LIN {X 0,Y 434.581,Z 927.636,A -85,B 0,C 180,E1 8882.861,E2 8882.861} C_VEL
LIN {X 0,Y 430.893,Z 955.392,A -85,B 0,C 180,E1 8887.344,E2 8887.344} C_VEL
LIN {X 0,Y 428.364,Z 976.944,A -85,B 0,C 180,E1 8892.013,E2 8892.013} C_VEL
LIN {X 0,Y 426.942,Z 993.408,A -85,B 0,C 180,E1 8896.966,E2 8896.966} C_VEL
LIN {X 0,Y 426.344,Z 1004.121,A -85,B 0,C 180,E1 8901.864,E2 8901.864} C_VEL
LIN {X 0,Y 426.1,Z 1008.94,A -85,B 0,C 180,E1 8905.941,E2 8905.941} C_VEL
LIN {X 0,Y 426.135,Z 1010.5,A -85,B 0,C 180,E1 8910.003,E2 8910.003} C_VEL
LIN {X 0,Y 426.114,Z 1008.916,A -85,B 0,C 180,E1 8914.065,E2 8914.065} C_VEL
LIN {X 0,Y 426.347,Z 1004.111,A -85,B 0,C 180,E1 8918.143,E2 8918.143} C_VEL
LIN {X 0,Y 427.008,Z 993.215,A -85,B 0,C 180,E1 8923.05,E2 8923.05} C_VEL
LIN {X 0,Y 428.484,Z 976.134,A -85,B 0,C 180,E1 8928.036,E2 8928.036} C_VEL
LIN {X 0,Y 430.871,Z 953.792,A -85,B 0,C 180,E1 8932.663,E2 8932.663} C_VEL
LIN {X 0,Y 434.231,Z 925.274,A -85,B 0,C 180,E1 8937.015,E2 8937.015} C_VEL
LIN {X 0,Y 438.15,Z 892.411,A -85,B 0,C 180,E1 8940.744,E2 8940.744} C_VEL
LIN {X 0,Y 442.235,Z 855.915,A -85,B 0,C 180,E1 8943.828,E2 8943.828} C_VEL
LIN {X 0,Y 446.217,Z 814.757,A -85,B 0,C 180,E1 8946.335,E2 8946.335} C_VEL
LIN {X 0,Y 449.648,Z 772.764,A -85,B 0,C 180,E1 8948.036,E2 8948.036} C_VEL
LIN {X 0,Y 450.402,Z 750.353,A -85,B 0,C 180,E1 8948.691,E2 8948.691} C_VEL
LIN {X 0,Y 439.584,Z 726.546,A -85,B 0,C 180,E1 8950.23,E2 8950.23} C_VEL
LIN {X 0,Y 430.713,Z 701.682,A -85,B 0,C 180,E1 8951.883,E2 8951.883} C_VEL
LIN {X 0,Y 424.876,Z 685.03,A -85,B 0,C 180,E1 8954.111,E2 8954.111} C_VEL
LIN {X 0,Y 424.882,Z 685.03,A -85,B 0,C 180,E1 8960.26,E2 8960.26} C_VEL
LIN {X 0,Y 424.85,Z 685.03,A -85,B 0,C 180,E1 8965.366,E2 8965.366} C_VEL
LIN {X 0,Y 424.908,Z 685.03,A -85,B 0,C 180,E1 8970.183,E2 8970.183} C_VEL
LIN {X 0,Y 425.058,Z 685.759,A -85,B 0,C 180,E1 8974.192,E2 8974.192} C_VEL
LIN {X 0,Y 435.61,Z 708.568,A -85,B 0,C 180,E1 8976.713,E2 8976.713} C_VEL
LIN {X 0,Y 439.993,Z 723.265,A -85,B 0,C 180,E1 8977.775,E2 8977.775} C_VEL
LIN {X 0,Y 437.409,Z 775.12,A -85,B 0,C 180,E1 8979.599,E2 8979.599} C_VEL
LIN {X 0,Y 435.839,Z 802.253,A -85,B 0,C 180,E1 8981.318,E2 8981.318} C_VEL
LIN {X 0,Y 433.74,Z 826.035,A -85,B 0,C 180,E1 8983.672,E2 8983.672} C_VEL
LIN {X 0,Y 431.655,Z 846.013,A -85,B 0,C 180,E1 8986.605,E2 8986.605} C_VEL
LIN {X 0,Y 429.88,Z 860.973,A -85,B 0,C 180,E1 8989.888,E2 8989.888} C_VEL
LIN {X 0,Y 428.712,Z 871.1,A -85,B 0,C 180,E1 8993.427,E2 8993.427} C_VEL
LIN {X 0,Y 428.238,Z 875.222,A -85,B 0,C 180,E1 8995.955,E2 8995.955} C_VEL
LIN {X 0,Y 427.911,Z 877.085,A -85,B 0,C 180,E1 8999.995,E2 8999.995} C_VEL
LIN {X 0,Y 427.908,Z 873.125,A -85,B 0,C 180,E1 9004.04,E2 9004.04} C_VEL
LIN {X 0,Y 428.392,Z 863.089,A -85,B 0,C 180,E1 9008.095,E2 9008.095} C_VEL
LIN {X 0,Y 429.506,Z 848.056,A -85,B 0,C 180,E1 9011.649,E2 9011.649} C_VEL
LIN {X 0,Y 431.114,Z 827.623,A -85,B 0,C 180,E1 9014.864,E2 9014.864} C_VEL
LIN {X 0,Y 432.915,Z 802.738,A -85,B 0,C 180,E1 9017.49,E2 9017.49} C_VEL
LIN {X 0,Y 434.545,Z 775.132,A -85,B 0,C 180,E1 9019.388,E2 9019.388} C_VEL
LIN {X 0,Y 435.512,Z 745.912,A -85,B 0,C 180,E1 9020.544,E2 9020.544} C_VEL
LIN {X 0,Y 435.429,Z 716.915,A -85,B 0,C 180,E1 9021.218,E2 9021.218} C_VEL
LIN {X 0,Y 425.206,Z 685.03,A -85,B 0,C 180,E1 9022.66,E2 9022.66} C_VEL
LIN {X 0,Y 424.891,Z 685.03,A -85,B 0,C 180,E1 9029.808,E2 9029.808} C_VEL
LIN {X 0,Y 424.913,Z 685.03,A -85,B 0,C 180,E1 9037.128,E2 9037.128} C_VEL
LIN {X 0,Y 424.882,Z 685.03,A -85,B 0,C 180,E1 9042.428,E2 9042.428} C_VEL
LIN {X 0,Y 424.889,Z 685.03,A -85,B 0,C 180,E1 9048.217,E2 9048.217} C_VEL
LIN {X 0,Y 424.853,Z 685.03,A -85,B 0,C 180,E1 9054.763,E2 9054.763} C_VEL
LIN {X 0,Y 425.044,Z 685.03,A -85,B 0,C 180,E1 9059.974,E2 9059.974} C_VEL
LIN {X 0,Y 438.959,Z 721.304,A -85,B 0,C 180,E1 9062.075,E2 9062.075} C_VEL
LIN {X 0,Y 441.889,Z 733.46,A -85,B 0,C 180,E1 9062.854,E2 9062.854} C_VEL
LIN {X 0,Y 439.577,Z 764.943,A -85,B 0,C 180,E1 9064.72,E2 9064.72} C_VEL
LIN {X 0,Y 436.7,Z 793.098,A -85,B 0,C 180,E1 9067.232,E2 9067.232} C_VEL
LIN {X 0,Y 433.564,Z 818.328,A -85,B 0,C 180,E1 9070.417,E2 9070.417} C_VEL
LIN {X 0,Y 430.741,Z 839.909,A -85,B 0,C 180,E1 9074.293,E2 9074.293} C_VEL
LIN {X 0,Y 428.905,Z 855.283,A -85,B 0,C 180,E1 9078.325,E2 9078.325} C_VEL
LIN {X 0,Y 427.683,Z 866.396,A -85,B 0,C 180,E1 9082.903,E2 9082.903} C_VEL
LIN {X 0,Y 427.355,Z 870.61,A -85,B 0,C 180,E1 9085.947,E2 9085.947} C_VEL
LIN {X 0,Y 427.257,Z 872.588,A -85,B 0,C 180,E1 9089.997,E2 9089.997} C_VEL
LIN {X 0,Y 427.468,Z 869.387,A -85,B 0,C 180,E1 9095.06,E2 9095.06} C_VEL
LIN {X 0,Y 428.256,Z 861.224,A -85,B 0,C 180,E1 9099.446,E2 9099.446} C_VEL
LIN {X 0,Y 429.883,Z 846.906,A -85,B 0,C 180,E1 9103.963,E2 9103.963} C_VEL
LIN {X 0,Y 432.277,Z 828.802,A -85,B 0,C 180,E1 9107.783,E2 9107.783} C_VEL
LIN {X 0,Y 435.266,Z 804.741,A -85,B 0,C 180,E1 9111.345,E2 9111.345} C_VEL
LIN {X 0,Y 438.411,Z 777.158,A -85,B 0,C 180,E1 9114.203,E2 9114.203} C_VEL
LIN {X 0,Y 441.046,Z 746.04,A -85,B 0,C 180,E1 9116.408,E2 9116.408} C_VEL
LIN {X 0,Y 441.406,Z 729.34,A -85,B 0,C 180,E1 9117.291,E2 9117.291} C_VEL
LIN {X 0,Y 430.11,Z 697.835,A -85,B 0,C 180,E1 9119.246,E2 9119.246} C_VEL
LIN {X 0,Y 425.006,Z 685.03,A -85,B 0,C 180,E1 9120.023,E2 9120.023} C_VEL
LIN {X 0,Y 424.844,Z 685.03,A -85,B 0,C 180,E1 9127.143,E2 9127.143} C_VEL
LIN {X 0,Y 424.822,Z 685.03,A -85,B 0,C 180,E1 9132.445,E2 9132.445} C_VEL
LIN {X 0,Y 424.867,Z 685.03,A -85,B 0,C 180,E1 9138.231,E2 9138.231} C_VEL
LIN {X 0,Y 424.852,Z 685.03,A -85,B 0,C 180,E1 9144.777,E2 9144.777} C_VEL
LIN {X 0,Y 424.934,Z 685.03,A -85,B 0,C 180,E1 9150.196,E2 9150.196} C_VEL
LIN {X 0,Y 425.242,Z 685.03,A -85,B 0,C 180,E1 9157.312,E2 9157.312} C_VEL
LIN {X 0,Y 425.495,Z 685.03,A -85,B 0,C 180,E1 9163.524,E2 9163.524} C_VEL
LIN {X 0,Y 425.69,Z 685.03,A -85,B 0,C 180,E1 9169.796,E2 9169.796} C_VEL
LIN {X 0,Y 425.89,Z 685.03,A -85,B 0,C 180,E1 9175.941,E2 9175.941} C_VEL
LIN {X 0,Y 426.083,Z 685.03,A -85,B 0,C 180,E1 9182.034,E2 9182.034} C_VEL
LIN {X 0,Y 425.686,Z 685.03,A -85,B 0,C 180,E1 9188.156,E2 9188.156} C_VEL
LIN {X 0,Y 425.437,Z 685.03,A -85,B 0,C 180,E1 9194.379,E2 9194.379} C_VEL
LIN {X 0,Y 425.24,Z 685.03,A -85,B 0,C 180,E1 9200.788,E2 9200.788} C_VEL
LIN {X 0,Y 424.989,Z 685.03,A -85,B 0,C 180,E1 9207.492,E2 9207.492} C_VEL
LIN {X 0,Y 424.842,Z 685.03,A -85,B 0,C 180,E1 9214.634,E2 9214.634} C_VEL
LIN {X 0,Y 424.88,Z 685.03,A -85,B 0,C 180,E1 9219.74,E2 9219.74} C_VEL
LIN {X 0,Y 424.929,Z 685.613,A -85,B 0,C 180,E1 9224.958,E2 9224.958} C_VEL
LIN {X 0,Y 435.905,Z 715.992,A -85,B 0,C 180,E1 9228.276,E2 9228.276} C_VEL
LIN {X 0,Y 453.307,Z 751.981,A -85,B 0,C 180,E1 9230.656,E2 9230.656} C_VEL
LIN {X 0,Y 451.051,Z 792.914,A -85,B 0,C 180,E1 9231.93,E2 9231.93} C_VEL
LIN {X 0,Y 447.298,Z 830.648,A -85,B 0,C 180,E1 9233.78,E2 9233.78} C_VEL
LIN {X 0,Y 442.865,Z 866.736,A -85,B 0,C 180,E1 9236.306,E2 9236.306} C_VEL
LIN {X 0,Y 438.213,Z 901.661,A -85,B 0,C 180,E1 9239.635,E2 9239.635} C_VEL
LIN {X 0,Y 434.581,Z 927.636,A -85,B 0,C 180,E1 9242.861,E2 9242.861} C_VEL
LIN {X 0,Y 429.124,Z 939.223,A -85,B 0,C 180,E1 9244.458,E2 9244.458} C_VEL
LIN {X 0,Y 423.822,Z 949.985,A -85,B 0,C 180,E1 9246.175,E2 9246.175} C_VEL
LIN {X 0,Y 421.006,Z 972.633,A -85,B 0,C 180,E1 9250.912,E2 9250.912} C_VEL
LIN {X 0,Y 419.279,Z 990.234,A -85,B 0,C 180,E1 9256,E2 9256} C_VEL
LIN {X 0,Y 418.584,Z 1001.205,A -85,B 0,C 180,E1 9260.667,E2 9260.667} C_VEL
LIN {X 0,Y 418.241,Z 1008.136,A -85,B 0,C 180,E1 9265.865,E2 9265.865} C_VEL
LIN {X 0,Y 418.261,Z 1009.846,A -85,B 0,C 180,E1 9270.003,E2 9270.003} C_VEL
LIN {X 0,Y 418.26,Z 1007.13,A -85,B 0,C 180,E1 9275.178,E2 9275.178} C_VEL
LIN {X 0,Y 418.604,Z 1000.03,A -85,B 0,C 180,E1 9279.863,E2 9279.863} C_VEL
LIN {X 0,Y 419.457,Z 987.963,A -85,B 0,C 180,E1 9284.59,E2 9284.59} C_VEL
LIN {X 0,Y 421.174,Z 970.321,A -85,B 0,C 180,E1 9289.359,E2 9289.359} C_VEL
LIN {X 0,Y 423.731,Z 947.19,A -85,B 0,C 180,E1 9293.894,E2 9293.894} C_VEL
LIN {X 0,Y 427.41,Z 917.918,A -85,B 0,C 180,E1 9298.154,E2 9298.154} C_VEL
LIN {X 0,Y 431.545,Z 883.702,A -85,B 0,C 180,E1 9301.873,E2 9301.873} C_VEL
LIN {X 0,Y 435.994,Z 844.862,A -85,B 0,C 180,E1 9304.982,E2 9304.982} C_VEL
LIN {X 0,Y 440.133,Z 803.438,A -85,B 0,C 180,E1 9307.337,E2 9307.337} C_VEL
LIN {X 0,Y 443.714,Z 760.178,A -85,B 0,C 180,E1 9308.928,E2 9308.928} C_VEL
LIN {X 0,Y 443.517,Z 753.15,A -85,B 0,C 180,E1 9309.172,E2 9309.172} C_VEL
LIN {X 0,Y 433.063,Z 728.03,A -85,B 0,C 180,E1 9310.864,E2 9310.864} C_VEL
LIN {X 0,Y 424.946,Z 704.873,A -85,B 0,C 180,E1 9312.523,E2 9312.523} C_VEL
LIN {X 0,Y 420.393,Z 694.266,A -85,B 0,C 180,E1 9313.748,E2 9313.748} C_VEL
LIN {X 0,Y 416.975,Z 685.03,A -85,B 0,C 180,E1 9315.334,E2 9315.334} C_VEL
LIN {X 0,Y 416.992,Z 685.03,A -85,B 0,C 180,E1 9322.032,E2 9322.032} C_VEL
LIN {X 0,Y 416.963,Z 685.03,A -85,B 0,C 180,E1 9329.556,E2 9329.556} C_VEL
LIN {X 0,Y 417.127,Z 685.437,A -85,B 0,C 180,E1 9332.851,E2 9332.851} C_VEL
LIN {X 0,Y 427.591,Z 707.36,A -85,B 0,C 180,E1 9335.736,E2 9335.736} C_VEL
LIN {X 0,Y 433.416,Z 725.205,A -85,B 0,C 180,E1 9337.233,E2 9337.233} C_VEL
LIN {X 0,Y 430.362,Z 778.741,A -85,B 0,C 180,E1 9339.25,E2 9339.25} C_VEL
LIN {X 0,Y 428.532,Z 806.342,A -85,B 0,C 180,E1 9341.121,E2 9341.121} C_VEL
LIN {X 0,Y 426.299,Z 829.518,A -85,B 0,C 180,E1 9343.547,E2 9343.547} C_VEL
LIN {X 0,Y 424.041,Z 849.221,A -85,B 0,C 180,E1 9346.622,E2 9346.622} C_VEL
LIN {X 0,Y 422.044,Z 864.475,A -85,B 0,C 180,E1 9350.218,E2 9350.218} C_VEL
LIN {X 0,Y 420.873,Z 873.677,A -85,B 0,C 180,E1 9353.821,E2 9353.821} C_VEL
LIN {X 0,Y 420.23,Z 878.301,A -85,B 0,C 180,E1 9357.938,E2 9357.938} C_VEL
LIN {X 0,Y 420.063,Z 877.143,A -85,B 0,C 180,E1 9362.054,E2 9362.054} C_VEL
LIN {X 0,Y 420.31,Z 870.117,A -85,B 0,C 180,E1 9366.178,E2 9366.178} C_VEL
LIN {X 0,Y 421.148,Z 857.596,A -85,B 0,C 180,E1 9370.021,E2 9370.021} C_VEL
LIN {X 0,Y 422.599,Z 840.277,A -85,B 0,C 180,E1 9373.415,E2 9373.415} C_VEL
LIN {X 0,Y 424.342,Z 818.559,A -85,B 0,C 180,E1 9376.324,E2 9376.324} C_VEL
LIN {X 0,Y 426.208,Z 792.037,A -85,B 0,C 180,E1 9378.708,E2 9378.708} C_VEL
LIN {X 0,Y 427.638,Z 763.471,A -85,B 0,C 180,E1 9380.319,E2 9380.319} C_VEL
LIN {X 0,Y 428.494,Z 727.084,A -85,B 0,C 180,E1 9381.351,E2 9381.351} C_VEL
LIN {X 0,Y 427.683,Z 717.143,A -85,B 0,C 180,E1 9381.629,E2 9381.629} C_VEL
LIN {X 0,Y 417.265,Z 685.03,A -85,B 0,C 180,E1 9383.061,E2 9383.061} C_VEL
LIN {X 0,Y 416.98,Z 685.03,A -85,B 0,C 180,E1 9390.432,E2 9390.432} C_VEL
LIN {X 0,Y 416.989,Z 685.03,A -85,B 0,C 180,E1 9397.956,E2 9397.956} C_VEL
LIN {X 0,Y 416.897,Z 685.03,A -85,B 0,C 180,E1 9403.613,E2 9403.613} C_VEL
LIN {X 0,Y 416.926,Z 685.03,A -85,B 0,C 180,E1 9409.457,E2 9409.457} C_VEL
LIN {X 0,Y 416.939,Z 685.03,A -85,B 0,C 180,E1 9414.608,E2 9414.608} C_VEL
LIN {X 0,Y 417.063,Z 685.03,A -85,B 0,C 180,E1 9419.329,E2 9419.329} C_VEL
LIN {X 0,Y 431.128,Z 720.992,A -85,B 0,C 180,E1 9421.458,E2 9421.458} C_VEL
LIN {X 0,Y 434.944,Z 734.898,A -85,B 0,C 180,E1 9422.397,E2 9422.397} C_VEL
LIN {X 0,Y 432.559,Z 766.155,A -85,B 0,C 180,E1 9424.281,E2 9424.281} C_VEL
LIN {X 0,Y 429.565,Z 794.116,A -85,B 0,C 180,E1 9426.808,E2 9426.808} C_VEL
LIN {X 0,Y 426.144,Z 820.08,A -85,B 0,C 180,E1 9430.146,E2 9430.146} C_VEL
LIN {X 0,Y 423.167,Z 841.477,A -85,B 0,C 180,E1 9434.081,E2 9434.081} C_VEL
LIN {X 0,Y 421.262,Z 856.527,A -85,B 0,C 180,E1 9438.11,E2 9438.11} C_VEL
LIN {X 0,Y 419.94,Z 867.642,A -85,B 0,C 180,E1 9442.771,E2 9442.771} C_VEL
LIN {X 0,Y 419.568,Z 871.858,A -85,B 0,C 180,E1 9445.872,E2 9445.872} C_VEL
LIN {X 0,Y 419.472,Z 873.833,A -85,B 0,C 180,E1 9449.997,E2 9449.997} C_VEL
LIN {X 0,Y 419.694,Z 870.635,A -85,B 0,C 180,E1 9455.154,E2 9455.154} C_VEL
LIN {X 0,Y 420.558,Z 862.472,A -85,B 0,C 180,E1 9459.62,E2 9459.62} C_VEL
LIN {X 0,Y 422.304,Z 848.154,A -85,B 0,C 180,E1 9464.218,E2 9464.218} C_VEL
LIN {X 0,Y 425.081,Z 828.545,A -85,B 0,C 180,E1 9468.362,E2 9468.362} C_VEL
LIN {X 0,Y 428.191,Z 804.977,A -85,B 0,C 180,E1 9471.851,E2 9471.851} C_VEL
LIN {X 0,Y 431.353,Z 778.059,A -85,B 0,C 180,E1 9474.657,E2 9474.657} C_VEL
LIN {X 0,Y 434.095,Z 747.258,A -85,B 0,C 180,E1 9476.864,E2 9476.864} C_VEL
LIN {X 0,Y 434.367,Z 731.277,A -85,B 0,C 180,E1 9477.739,E2 9477.739} C_VEL
LIN {X 0,Y 423.213,Z 700.221,A -85,B 0,C 180,E1 9479.74,E2 9479.74} C_VEL
LIN {X 0,Y 417.086,Z 685.03,A -85,B 0,C 180,E1 9480.631,E2 9480.631} C_VEL
LIN {X 0,Y 416.91,Z 685.03,A -85,B 0,C 180,E1 9487.973,E2 9487.973} C_VEL
LIN {X 0,Y 416.848,Z 685.03,A -85,B 0,C 180,E1 9493.626,E2 9493.626} C_VEL
LIN {X 0,Y 416.908,Z 685.03,A -85,B 0,C 180,E1 9499.471,E2 9499.471} C_VEL
LIN {X 0,Y 416.938,Z 685.03,A -85,B 0,C 180,E1 9504.623,E2 9504.623} C_VEL
LIN {X 0,Y 417.038,Z 685.03,A -85,B 0,C 180,E1 9511.948,E2 9511.948} C_VEL
LIN {X 0,Y 417.345,Z 685.03,A -85,B 0,C 180,E1 9518.81,E2 9518.81} C_VEL
LIN {X 0,Y 417.681,Z 685.03,A -85,B 0,C 180,E1 9525.357,E2 9525.357} C_VEL
LIN {X 0,Y 417.788,Z 685.03,A -85,B 0,C 180,E1 9531.698,E2 9531.698} C_VEL
LIN {X 0,Y 418.033,Z 685.03,A -85,B 0,C 180,E1 9537.936,E2 9537.936} C_VEL
LIN {X 0,Y 417.941,Z 685.03,A -85,B 0,C 180,E1 9544.145,E2 9544.145} C_VEL
LIN {X 0,Y 417.641,Z 685.03,A -85,B 0,C 180,E1 9550.412,E2 9550.412} C_VEL
LIN {X 0,Y 417.437,Z 685.03,A -85,B 0,C 180,E1 9556.813,E2 9556.813} C_VEL
LIN {X 0,Y 417.189,Z 685.03,A -85,B 0,C 180,E1 9563.448,E2 9563.448} C_VEL
LIN {X 0,Y 416.97,Z 685.03,A -85,B 0,C 180,E1 9570.444,E2 9570.444} C_VEL
LIN {X 0,Y 416.993,Z 685.03,A -85,B 0,C 180,E1 9577.968,E2 9577.968} C_VEL
LIN {X 0,Y 416.96,Z 685.716,A -85,B 0,C 180,E1 9584.179,E2 9584.179} C_VEL
LIN {X 0,Y 427.816,Z 715.235,A -85,B 0,C 180,E1 9587.487,E2 9587.487} C_VEL
LIN {X 0,Y 447.114,Z 756.966,A -85,B 0,C 180,E1 9590.254,E2 9590.254} C_VEL
LIN {X 0,Y 443.634,Z 799.853,A -85,B 0,C 180,E1 9591.689,E2 9591.689} C_VEL
LIN {X 0,Y 439.228,Z 839.677,A -85,B 0,C 180,E1 9593.854,E2 9593.854} C_VEL
LIN {X 0,Y 434.278,Z 876.572,A -85,B 0,C 180,E1 9596.723,E2 9596.723} C_VEL
LIN {X 0,Y 429.369,Z 910.527,A -85,B 0,C 180,E1 9600.311,E2 9600.311} C_VEL
LIN {X 0,Y 424.995,Z 941.035,A -85,B 0,C 180,E1 9604.633,E2 9604.633} C_VEL
LIN {X 0,Y 423.822,Z 949.985,A -85,B 0,C 180,E1 9606.175,E2 9606.175} C_VEL
LIN {X 0,Y 418.537,Z 959.925,A -85,B 0,C 180,E1 9608.012,E2 9608.012} C_VEL
LIN {X 0,Y 413.58,Z 968.967,A -85,B 0,C 180,E1 9609.965,E2 9609.965} C_VEL
LIN {X 0,Y 411.62,Z 987.327,A -85,B 0,C 180,E1 9615.133,E2 9615.133} C_VEL
LIN {X 0,Y 410.755,Z 1000.089,A -85,B 0,C 180,E1 9620.487,E2 9620.487} C_VEL
LIN {X 0,Y 410.416,Z 1007.046,A -85,B 0,C 180,E1 9625.786,E2 9625.786} C_VEL
LIN {X 0,Y 410.44,Z 1008.743,A -85,B 0,C 180,E1 9630.003,E2 9630.003} C_VEL
LIN {X 0,Y 410.467,Z 1005.955,A -85,B 0,C 180,E1 9635.277,E2 9635.277} C_VEL
LIN {X 0,Y 410.785,Z 998.736,A -85,B 0,C 180,E1 9640.053,E2 9640.053} C_VEL
LIN {X 0,Y 411.646,Z 986.479,A -85,B 0,C 180,E1 9644.873,E2 9644.873} C_VEL
LIN {X 0,Y 413.405,Z 968.559,A -85,B 0,C 180,E1 9649.738,E2 9649.738} C_VEL
LIN {X 0,Y 416.138,Z 945.12,A -85,B 0,C 180,E1 9654.353,E2 9654.353} C_VEL
LIN {X 0,Y 419.799,Z 916.534,A -85,B 0,C 180,E1 9658.551,E2 9658.551} C_VEL
LIN {X 0,Y 424.244,Z 881.946,A -85,B 0,C 180,E1 9662.361,E2 9662.361} C_VEL
LIN {X 0,Y 428.916,Z 843.014,A -85,B 0,C 180,E1 9665.523,E2 9665.523} C_VEL
LIN {X 0,Y 433.342,Z 801.026,A -85,B 0,C 180,E1 9667.946,E2 9667.946} C_VEL
LIN {X 0,Y 436.927,Z 756.261,A -85,B 0,C 180,E1 9669.64,E2 9669.64} C_VEL
LIN {X 0,Y 427.136,Z 731.026,A -85,B 0,C 180,E1 9671.441,E2 9671.441} C_VEL
LIN {X 0,Y 419.894,Z 709.414,A -85,B 0,C 180,E1 9673.071,E2 9673.071} C_VEL
LIN {X 0,Y 411.681,Z 692.09,A -85,B 0,C 180,E1 9675.255,E2 9675.255} C_VEL
LIN {X 0,Y 409.017,Z 685.03,A -85,B 0,C 180,E1 9676.586,E2 9676.586} C_VEL
LIN {X 0,Y 409.035,Z 685.03,A -85,B 0,C 180,E1 9683.822,E2 9683.822} C_VEL
LIN {X 0,Y 409.077,Z 685.058,A -85,B 0,C 180,E1 9691.144,E2 9691.144} C_VEL
LIN {X 0,Y 410.65,Z 689.708,A -85,B 0,C 180,E1 9691.887,E2 9691.887} C_VEL
LIN {X 0,Y 413.732,Z 694.843,A -85,B 0,C 180,E1 9692.89,E2 9692.89} C_VEL
LIN {X 0,Y 421.77,Z 711.103,A -85,B 0,C 180,E1 9695.192,E2 9695.192} C_VEL
LIN {X 0,Y 426.973,Z 727.204,A -85,B 0,C 180,E1 9696.659,E2 9696.659} C_VEL
LIN {X 0,Y 423.424,Z 781.346,A -85,B 0,C 180,E1 9698.828,E2 9698.828} C_VEL
LIN {X 0,Y 421.359,Z 809.012,A -85,B 0,C 180,E1 9700.787,E2 9700.787} C_VEL
LIN {X 0,Y 419.016,Z 831.698,A -85,B 0,C 180,E1 9703.252,E2 9703.252} C_VEL
LIN {X 0,Y 416.602,Z 851.129,A -85,B 0,C 180,E1 9706.379,E2 9706.379} C_VEL
LIN {X 0,Y 414.445,Z 866.177,A -85,B 0,C 180,E1 9710.037,E2 9710.037} C_VEL
LIN {X 0,Y 413.194,Z 875.237,A -85,B 0,C 180,E1 9713.706,E2 9713.706} C_VEL
LIN {X 0,Y 412.474,Z 879.735,A -85,B 0,C 180,E1 9717.899,E2 9717.899} C_VEL
LIN {X 0,Y 412.299,Z 878.443,A -85,B 0,C 180,E1 9722.093,E2 9722.093} C_VEL
LIN {X 0,Y 412.555,Z 871.294,A -85,B 0,C 180,E1 9726.295,E2 9726.295} C_VEL
LIN {X 0,Y 413.433,Z 858.827,A -85,B 0,C 180,E1 9730.163,E2 9730.163} C_VEL
LIN {X 0,Y 414.951,Z 841.191,A -85,B 0,C 180,E1 9733.667,E2 9733.667} C_VEL
LIN {X 0,Y 416.822,Z 819.344,A -85,B 0,C 180,E1 9736.627,E2 9736.627} C_VEL
LIN {X 0,Y 418.778,Z 792.638,A -85,B 0,C 180,E1 9739.053,E2 9739.053} C_VEL
LIN {X 0,Y 420.233,Z 764.607,A -85,B 0,C 180,E1 9740.659,E2 9740.659} C_VEL
LIN {X 0,Y 421.194,Z 726.518,A -85,B 0,C 180,E1 9741.759,E2 9741.759} C_VEL
LIN {X 0,Y 419.368,Z 715.746,A -85,B 0,C 180,E1 9742.125,E2 9742.125} C_VEL
LIN {X 0,Y 409.293,Z 685.03,A -85,B 0,C 180,E1 9743.613,E2 9743.613} C_VEL
LIN {X 0,Y 409.071,Z 685.03,A -85,B 0,C 180,E1 9748.648,E2 9748.648} C_VEL
LIN {X 0,Y 409.039,Z 685.03,A -85,B 0,C 180,E1 9756.166,E2 9756.166} C_VEL
LIN {X 0,Y 408.9,Z 685.03,A -85,B 0,C 180,E1 9762.424,E2 9762.424} C_VEL
LIN {X 0,Y 408.899,Z 685.03,A -85,B 0,C 180,E1 9768.367,E2 9768.367} C_VEL
LIN {X 0,Y 409.045,Z 685.03,A -85,B 0,C 180,E1 9774.238,E2 9774.238} C_VEL
LIN {X 0,Y 409.177,Z 685.48,A -85,B 0,C 180,E1 9778.668,E2 9778.668} C_VEL
LIN {X 0,Y 423.38,Z 720.591,A -85,B 0,C 180,E1 9780.817,E2 9780.817} C_VEL
LIN {X 0,Y 427.988,Z 737.484,A -85,B 0,C 180,E1 9781.984,E2 9781.984} C_VEL
LIN {X 0,Y 425.4,Z 769.044,A -85,B 0,C 180,E1 9783.957,E2 9783.957} C_VEL
LIN {X 0,Y 422.114,Z 797.725,A -85,B 0,C 180,E1 9786.651,E2 9786.651} C_VEL
LIN {X 0,Y 418.68,Z 822.2,A -85,B 0,C 180,E1 9789.924,E2 9789.924} C_VEL
LIN {X 0,Y 415.6,Z 843.054,A -85,B 0,C 180,E1 9793.863,E2 9793.863} C_VEL
LIN {X 0,Y 413.389,Z 859.359,A -85,B 0,C 180,E1 9798.414,E2 9798.414} C_VEL
LIN {X 0,Y 412.204,Z 868.887,A -85,B 0,C 180,E1 9802.635,E2 9802.635} C_VEL
LIN {X 0,Y 411.79,Z 873.104,A -85,B 0,C 180,E1 9805.794,E2 9805.794} C_VEL
LIN {X 0,Y 411.688,Z 875.077,A -85,B 0,C 180,E1 9809.997,E2 9809.997} C_VEL
LIN {X 0,Y 411.919,Z 871.884,A -85,B 0,C 180,E1 9815.252,E2 9815.252} C_VEL
LIN {X 0,Y 412.925,Z 863.069,A -85,B 0,C 180,E1 9820.081,E2 9820.081} C_VEL
LIN {X 0,Y 414.729,Z 849.403,A -85,B 0,C 180,E1 9824.484,E2 9824.484} C_VEL
LIN {X 0,Y 417.68,Z 829.79,A -85,B 0,C 180,E1 9828.699,E2 9828.699} C_VEL
LIN {X 0,Y 420.965,Z 806.217,A -85,B 0,C 180,E1 9832.246,E2 9832.246} C_VEL
LIN {X 0,Y 424.282,Z 779.206,A -85,B 0,C 180,E1 9835.104,E2 9835.104} C_VEL
LIN {X 0,Y 427.167,Z 748.477,A -85,B 0,C 180,E1 9837.336,E2 9837.336} C_VEL
LIN {X 0,Y 427.657,Z 734.346,A -85,B 0,C 180,E1 9838.118,E2 9838.118} C_VEL
LIN {X 0,Y 416.856,Z 703.699,A -85,B 0,C 180,E1 9840.179,E2 9840.179} C_VEL
LIN {X 0,Y 409.169,Z 685.03,A -85,B 0,C 180,E1 9841.315,E2 9841.315} C_VEL
LIN {X 0,Y 408.994,Z 685.03,A -85,B 0,C 180,E1 9846.178,E2 9846.178} C_VEL
LIN {X 0,Y 408.844,Z 685.03,A -85,B 0,C 180,E1 9852.436,E2 9852.436} C_VEL
LIN {X 0,Y 408.877,Z 685.03,A -85,B 0,C 180,E1 9858.381,E2 9858.381} C_VEL
LIN {X 0,Y 409.042,Z 685.03,A -85,B 0,C 180,E1 9864.252,E2 9864.252} C_VEL
LIN {X 0,Y 409.101,Z 685.03,A -85,B 0,C 180,E1 9871.354,E2 9871.354} C_VEL
LIN {X 0,Y 409.373,Z 685.03,A -85,B 0,C 180,E1 9878.377,E2 9878.377} C_VEL
LIN {X 0,Y 409.729,Z 685.03,A -85,B 0,C 180,E1 9885.066,E2 9885.066} C_VEL
LIN {X 0,Y 409.895,Z 685.03,A -85,B 0,C 180,E1 9891.537,E2 9891.537} C_VEL
LIN {X 0,Y 410.126,Z 685.03,A -85,B 0,C 180,E1 9897.896,E2 9897.896} C_VEL
LIN {X 0,Y 410.029,Z 685.03,A -85,B 0,C 180,E1 9904.225,E2 9904.225} C_VEL
LIN {X 0,Y 409.736,Z 685.03,A -85,B 0,C 180,E1 9910.615,E2 9910.615} C_VEL
LIN {X 0,Y 409.513,Z 685.03,A -85,B 0,C 180,E1 9917.148,E2 9917.148} C_VEL
LIN {X 0,Y 409.247,Z 685.03,A -85,B 0,C 180,E1 9923.932,E2 9923.932} C_VEL
LIN {X 0,Y 408.972,Z 685.03,A -85,B 0,C 180,E1 9931.105,E2 9931.105} C_VEL
LIN {X 0,Y 409.037,Z 685.03,A -85,B 0,C 180,E1 9936.178,E2 9936.178} C_VEL
LIN {X 0,Y 409.027,Z 685.523,A -85,B 0,C 180,E1 9943.348,E2 9943.348} C_VEL
LIN {X 0,Y 419.701,Z 714.419,A -85,B 0,C 180,E1 9946.67,E2 9946.67} C_VEL
LIN {X 0,Y 440.299,Z 760.438,A -85,B 0,C 180,E1 9949.779,E2 9949.779} C_VEL
LIN {X 0,Y 436.85,Z 800.129,A -85,B 0,C 180,E1 9951.166,E2 9951.166} C_VEL
LIN {X 0,Y 432.303,Z 839.056,A -85,B 0,C 180,E1 9953.323,E2 9953.323} C_VEL
LIN {X 0,Y 427.241,Z 875.203,A -85,B 0,C 180,E1 9956.166,E2 9956.166} C_VEL
LIN {X 0,Y 422.069,Z 909.295,A -85,B 0,C 180,E1 9959.807,E2 9959.807} C_VEL
LIN {X 0,Y 417.59,Z 938.768,A -85,B 0,C 180,E1 9964.016,E2 9964.016} C_VEL
LIN {X 0,Y 414.25,Z 963.172,A -85,B 0,C 180,E1 9968.639,E2 9968.639} C_VEL
LIN {X 0,Y 413.58,Z 968.967,A -85,B 0,C 180,E1 9969.965,E2 9969.965} C_VEL
LIN {X 0,Y 410.401,Z 975.191,A -85,B 0,C 180,E1 9971.513,E2 9971.513} C_VEL
LIN {X 0,Y 404.146,Z 983.335,A -85,B 0,C 180,E1 9973.908,E2 9973.908} C_VEL
LIN {X 0,Y 403.982,Z 984.215,A -85,B 0,C 180,E1 9974.192,E2 9974.192} C_VEL
LIN {X 0,Y 403.004,Z 997.99,A -85,B 0,C 180,E1 9979.758,E2 9979.758} C_VEL
LIN {X 0,Y 402.604,Z 1005.001,A -85,B 0,C 180,E1 9984.626,E2 9984.626} C_VEL
LIN {X 0,Y 402.616,Z 1007.64,A -85,B 0,C 180,E1 9990.003,E2 9990.003} C_VEL
LIN {X 0,Y 402.653,Z 1004.777,A -85,B 0,C 180,E1 9995.38,E2 9995.38} C_VEL
LIN {X 0,Y 402.973,Z 997.439,A -85,B 0,C 180,E1 10000.25,E2 10000.25} C_VEL
LIN {X 0,Y 403.874,Z 985.008,A -85,B 0,C 180,E1 10005.166,E2 10005.166} C_VEL
LIN {X 0,Y 405.691,Z 966.805,A -85,B 0,C 180,E1 10010.129,E2 10010.129} C_VEL
LIN {X 0,Y 408.728,Z 942.214,A -85,B 0,C 180,E1 10014.964,E2 10014.964} C_VEL
LIN {X 0,Y 412.633,Z 912.622,A -85,B 0,C 180,E1 10019.288,E2 10019.288} C_VEL
LIN {X 0,Y 417.159,Z 878.702,A -85,B 0,C 180,E1 10023.018,E2 10023.018} C_VEL
LIN {X 0,Y 422.099,Z 839.703,A -85,B 0,C 180,E1 10026.196,E2 10026.196} C_VEL
LIN {X 0,Y 426.927,Z 796.677,A -85,B 0,C 180,E1 10028.682,E2 10028.682} C_VEL
LIN {X 0,Y 430.27,Z 759.138,A -85,B 0,C 180,E1 10030.154,E2 10030.154} C_VEL
LIN {X 0,Y 420.632,Z 731.385,A -85,B 0,C 180,E1 10032.222,E2 10032.222} C_VEL
LIN {X 0,Y 413.804,Z 711.142,A -85,B 0,C 180,E1 10033.947,E2 10033.947} C_VEL
LIN {X 0,Y 406.131,Z 695.27,A -85,B 0,C 180,E1 10036.21,E2 10036.21} C_VEL
LIN {X 0,Y 402.659,Z 689.814,A -85,B 0,C 180,E1 10037.475,E2 10037.475} C_VEL
LIN {X 0,Y 401.039,Z 685.03,A -85,B 0,C 180,E1 10038.528,E2 10038.528} C_VEL
LIN {X 0,Y 401.069,Z 685.03,A -85,B 0,C 180,E1 10045.877,E2 10045.877} C_VEL
LIN {X 0,Y 401.085,Z 685.464,A -85,B 0,C 180,E1 10048.882,E2 10048.882} C_VEL
LIN {X 0,Y 408.554,Z 698.82,A -85,B 0,C 180,E1 10052.176,E2 10052.176} C_VEL
LIN {X 0,Y 417.146,Z 717.732,A -85,B 0,C 180,E1 10054.952,E2 10054.952} C_VEL
LIN {X 0,Y 420.523,Z 730.232,A -85,B 0,C 180,E1 10056.084,E2 10056.084} C_VEL
LIN {X 0,Y 416.544,Z 784.092,A -85,B 0,C 180,E1 10058.386,E2 10058.386} C_VEL
LIN {X 0,Y 414.243,Z 811.827,A -85,B 0,C 180,E1 10060.444,E2 10060.444} C_VEL
LIN {X 0,Y 411.541,Z 835.812,A -85,B 0,C 180,E1 10063.213,E2 10063.213} C_VEL
LIN {X 0,Y 408.977,Z 854.397,A -85,B 0,C 180,E1 10066.392,E2 10066.392} C_VEL
LIN {X 0,Y 406.848,Z 868.085,A -85,B 0,C 180,E1 10069.909,E2 10069.909} C_VEL
LIN {X 0,Y 405.517,Z 876.821,A -85,B 0,C 180,E1 10073.586,E2 10073.586} C_VEL
LIN {X 0,Y 404.731,Z 881.181,A -85,B 0,C 180,E1 10077.859,E2 10077.859} C_VEL
LIN {X 0,Y 404.534,Z 879.747,A -85,B 0,C 180,E1 10082.133,E2 10082.133} C_VEL
LIN {X 0,Y 404.778,Z 872.463,A -85,B 0,C 180,E1 10086.416,E2 10086.416} C_VEL
LIN {X 0,Y 405.681,Z 860.343,A -85,B 0,C 180,E1 10090.236,E2 10090.236} C_VEL
LIN {X 0,Y 407.306,Z 842.043,A -85,B 0,C 180,E1 10093.928,E2 10093.928} C_VEL
LIN {X 0,Y 409.308,Z 819.566,A -85,B 0,C 180,E1 10096.993,E2 10096.993} C_VEL
LIN {X 0,Y 411.311,Z 793.261,A -85,B 0,C 180,E1 10099.4,E2 10099.4} C_VEL
LIN {X 0,Y 412.908,Z 763.731,A -85,B 0,C 180,E1 10101.092,E2 10101.092} C_VEL
LIN {X 0,Y 413.425,Z 721.893,A -85,B 0,C 180,E1 10102.31,E2 10102.31} C_VEL
LIN {X 0,Y 401.338,Z 685.03,A -85,B 0,C 180,E1 10104.05,E2 10104.05} C_VEL
LIN {X 0,Y 401.084,Z 685.03,A -85,B 0,C 180,E1 10111.776,E2 10111.776} C_VEL
LIN {X 0,Y 401.024,Z 685.03,A -85,B 0,C 180,E1 10117.786,E2 10117.786} C_VEL
LIN {X 0,Y 400.989,Z 685.03,A -85,B 0,C 180,E1 10124.348,E2 10124.348} C_VEL
LIN {X 0,Y 400.998,Z 685.03,A -85,B 0,C 180,E1 10130.222,E2 10130.222} C_VEL
LIN {X 0,Y 401.205,Z 685.594,A -85,B 0,C 180,E1 10137.948,E2 10137.948} C_VEL
LIN {X 0,Y 416.148,Z 721.645,A -85,B 0,C 180,E1 10140.252,E2 10140.252} C_VEL
LIN {X 0,Y 421.028,Z 740.077,A -85,B 0,C 180,E1 10141.556,E2 10141.556} C_VEL
LIN {X 0,Y 418.19,Z 771.889,A -85,B 0,C 180,E1 10143.617,E2 10143.617} C_VEL
LIN {X 0,Y 414.781,Z 800.526,A -85,B 0,C 180,E1 10146.405,E2 10146.405} C_VEL
LIN {X 0,Y 410.974,Z 826.085,A -85,B 0,C 180,E1 10149.979,E2 10149.979} C_VEL
LIN {X 0,Y 407.819,Z 845.908,A -85,B 0,C 180,E1 10153.94,E2 10153.94} C_VEL
LIN {X 0,Y 405.742,Z 860.604,A -85,B 0,C 180,E1 10158.193,E2 10158.193} C_VEL
LIN {X 0,Y 404.474,Z 870.132,A -85,B 0,C 180,E1 10162.493,E2 10162.493} C_VEL
LIN {X 0,Y 404.006,Z 874.351,A -85,B 0,C 180,E1 10165.712,E2 10165.712} C_VEL
LIN {X 0,Y 403.907,Z 876.322,A -85,B 0,C 180,E1 10169.997,E2 10169.997} C_VEL
LIN {X 0,Y 404.148,Z 873.132,A -85,B 0,C 180,E1 10175.353,E2 10175.353} C_VEL
LIN {X 0,Y 405.187,Z 864.797,A -85,B 0,C 180,E1 10180.064,E2 10180.064} C_VEL
LIN {X 0,Y 407.15,Z 850.655,A -85,B 0,C 180,E1 10184.759,E2 10184.759} C_VEL
LIN {X 0,Y 410.285,Z 831.036,A -85,B 0,C 180,E1 10189.049,E2 10189.049} C_VEL
LIN {X 0,Y 413.773,Z 807.455,A -85,B 0,C 180,E1 10192.654,E2 10192.654} C_VEL
LIN {X 0,Y 417.276,Z 779.998,A -85,B 0,C 180,E1 10195.599,E2 10195.599} C_VEL
LIN {X 0,Y 420.257,Z 749.699,A -85,B 0,C 180,E1 10197.824,E2 10197.824} C_VEL
LIN {X 0,Y 420.71,Z 736.435,A -85,B 0,C 180,E1 10198.577,E2 10198.577} C_VEL
LIN {X 0,Y 409.812,Z 705.312,A -85,B 0,C 180,E1 10200.743,E2 10200.743} C_VEL
LIN {X 0,Y 401.211,Z 685.03,A -85,B 0,C 180,E1 10201.999,E2 10201.999} C_VEL
LIN {X 0,Y 400.936,Z 685.03,A -85,B 0,C 180,E1 10209.777,E2 10209.777} C_VEL
LIN {X 0,Y 400.955,Z 685.03,A -85,B 0,C 180,E1 10215.647,E2 10215.647} C_VEL
LIN {X 0,Y 401.002,Z 685.03,A -85,B 0,C 180,E1 10222.99,E2 10222.99} C_VEL
LIN {X 0,Y 401.075,Z 685.03,A -85,B 0,C 180,E1 10229.921,E2 10229.921} C_VEL
LIN {X 0,Y 401.299,Z 685.03,A -85,B 0,C 180,E1 10235.574,E2 10235.574} C_VEL
LIN {X 0,Y 401.664,Z 685.03,A -85,B 0,C 180,E1 10242.516,E2 10242.516} C_VEL
LIN {X 0,Y 401.923,Z 685.03,A -85,B 0,C 180,E1 10249.186,E2 10249.186} C_VEL
LIN {X 0,Y 402.165,Z 685.03,A -85,B 0,C 180,E1 10255.701,E2 10255.701} C_VEL
LIN {X 0,Y 402.392,Z 685.03,A -85,B 0,C 180,E1 10262.154,E2 10262.154} C_VEL
LIN {X 0,Y 401.898,Z 685.03,A -85,B 0,C 180,E1 10268.642,E2 10268.642} C_VEL
LIN {X 0,Y 401.661,Z 685.03,A -85,B 0,C 180,E1 10275.251,E2 10275.251} C_VEL
LIN {X 0,Y 401.394,Z 685.03,A -85,B 0,C 180,E1 10282.086,E2 10282.086} C_VEL
LIN {X 0,Y 401.064,Z 685.03,A -85,B 0,C 180,E1 10289.286,E2 10289.286} C_VEL
LIN {X 0,Y 401.045,Z 685.03,A -85,B 0,C 180,E1 10294.363,E2 10294.363} C_VEL
LIN {X 0,Y 400.974,Z 685.03,A -85,B 0,C 180,E1 10301.18,E2 10301.18} C_VEL
LIN {X 0,Y 401.07,Z 685.709,A -85,B 0,C 180,E1 10302.533,E2 10302.533} C_VEL
LIN {X 0,Y 411.289,Z 713.116,A -85,B 0,C 180,E1 10305.792,E2 10305.792} C_VEL
LIN {X 0,Y 433.477,Z 761.48,A -85,B 0,C 180,E1 10309.215,E2 10309.215} C_VEL
LIN {X 0,Y 429.85,Z 802.028,A -85,B 0,C 180,E1 10310.712,E2 10310.712} C_VEL
LIN {X 0,Y 425.063,Z 840.789,A -85,B 0,C 180,E1 10312.941,E2 10312.941} C_VEL
LIN {X 0,Y 419.747,Z 876.791,A -85,B 0,C 180,E1 10315.874,E2 10315.874} C_VEL
LIN {X 0,Y 414.323,Z 910.898,A -85,B 0,C 180,E1 10319.648,E2 10319.648} C_VEL
LIN {X 0,Y 409.569,Z 940.785,A -85,B 0,C 180,E1 10324.1,E2 10324.1} C_VEL
LIN {X 0,Y 406.078,Z 965.477,A -85,B 0,C 180,E1 10329.045,E2 10329.045} C_VEL
LIN {X 0,Y 403.982,Z 984.215,A -85,B 0,C 180,E1 10334.192,E2 10334.192} C_VEL
LIN {X 0,Y 401.07,Z 988.977,A -85,B 0,C 180,E1 10335.884,E2 10335.884} C_VEL
LIN {X 0,Y 395.342,Z 994.767,A -85,B 0,C 180,E1 10338.496,E2 10338.496} C_VEL
LIN {X 0,Y 395.23,Z 995.373,A -85,B 0,C 180,E1 10338.802,E2 10338.802} C_VEL
LIN {X 0,Y 394.858,Z 1002.862,A -85,B 0,C 180,E1 10343.526,E2 10343.526} C_VEL
LIN {X 0,Y 394.752,Z 1006.141,A -85,B 0,C 180,E1 10347.812,E2 10347.812} C_VEL
LIN {X 0,Y 394.803,Z 1006.033,A -85,B 0,C 180,E1 10352.194,E2 10352.194} C_VEL
LIN {X 0,Y 395.005,Z 1000.86,A -85,B 0,C 180,E1 10357.688,E2 10357.688} C_VEL
LIN {X 0,Y 395.503,Z 991.223,A -85,B 0,C 180,E1 10362.677,E2 10362.677} C_VEL
LIN {X 0,Y 396.987,Z 974.605,A -85,B 0,C 180,E1 10368.142,E2 10368.142} C_VEL
LIN {X 0,Y 399.488,Z 953.18,A -85,B 0,C 180,E1 10373.078,E2 10373.078} C_VEL
LIN {X 0,Y 403.195,Z 925.233,A -85,B 0,C 180,E1 10377.823,E2 10377.823} C_VEL
LIN {X 0,Y 407.82,Z 892.58,A -85,B 0,C 180,E1 10381.958,E2 10381.958} C_VEL
LIN {X 0,Y 413.194,Z 853.841,A -85,B 0,C 180,E1 10385.598,E2 10385.598} C_VEL
LIN {X 0,Y 418.347,Z 813.286,A -85,B 0,C 180,E1 10388.365,E2 10388.365} C_VEL
LIN {X 0,Y 423.132,Z 771.668,A -85,B 0,C 180,E1 10390.309,E2 10390.309} C_VEL
LIN {X 0,Y 423.334,Z 760.95,A -85,B 0,C 180,E1 10390.775,E2 10390.775} C_VEL
LIN {X 0,Y 414.383,Z 731.708,A -85,B 0,C 180,E1 10393.063,E2 10393.063} C_VEL
LIN {X 0,Y 407.904,Z 712.926,A -85,B 0,C 180,E1 10394.909,E2 10394.909} C_VEL
LIN {X 0,Y 400.947,Z 698.091,A -85,B 0,C 180,E1 10397.354,E2 10397.354} C_VEL
LIN {X 0,Y 397.299,Z 692.007,A -85,B 0,C 180,E1 10399.113,E2 10399.113} C_VEL
LIN {X 0,Y 393.415,Z 687.071,A -85,B 0,C 180,E1 10403.004,E2 10403.004} C_VEL
LIN {X 0,Y 394.428,Z 689.369,A -85,B 0,C 180,E1 10406.246,E2 10406.246} C_VEL
LIN {X 0,Y 397.739,Z 692.568,A -85,B 0,C 180,E1 10408.54,E2 10408.54} C_VEL
LIN {X 0,Y 404.286,Z 704.839,A -85,B 0,C 180,E1 10411.769,E2 10411.769} C_VEL
LIN {X 0,Y 411.896,Z 722.603,A -85,B 0,C 180,E1 10414.494,E2 10414.494} C_VEL
LIN {X 0,Y 414.474,Z 731.609,A -85,B 0,C 180,E1 10415.411,E2 10415.411} C_VEL
LIN {X 0,Y 409.789,Z 786.141,A -85,B 0,C 180,E1 10417.88,E2 10417.88} C_VEL
LIN {X 0,Y 407.318,Z 813.321,A -85,B 0,C 180,E1 10419.956,E2 10419.956} C_VEL
LIN {X 0,Y 404.534,Z 836.297,A -85,B 0,C 180,E1 10422.634,E2 10422.634} C_VEL
LIN {X 0,Y 401.554,Z 856.399,A -85,B 0,C 180,E1 10426.135,E2 10426.135} C_VEL
LIN {X 0,Y 399.066,Z 871.055,A -85,B 0,C 180,E1 10430.134,E2 10430.134} C_VEL
LIN {X 0,Y 397.841,Z 878.418,A -85,B 0,C 180,E1 10433.462,E2 10433.462} C_VEL
LIN {X 0,Y 396.975,Z 882.633,A -85,B 0,C 180,E1 10437.817,E2 10437.817} C_VEL
LIN {X 0,Y 396.767,Z 881.038,A -85,B 0,C 180,E1 10442.175,E2 10442.175} C_VEL
LIN {X 0,Y 397.023,Z 873.624,A -85,B 0,C 180,E1 10446.542,E2 10446.542} C_VEL
LIN {X 0,Y 398.047,Z 860.451,A -85,B 0,C 180,E1 10450.656,E2 10450.656} C_VEL
LIN {X 0,Y 399.701,Z 842.893,A -85,B 0,C 180,E1 10454.199,E2 10454.199} C_VEL
LIN {X 0,Y 401.822,Z 819.827,A -85,B 0,C 180,E1 10457.363,E2 10457.363} C_VEL
LIN {X 0,Y 403.867,Z 793.79,A -85,B 0,C 180,E1 10459.765,E2 10459.765} C_VEL
LIN {X 0,Y 405.499,Z 764.638,A -85,B 0,C 180,E1 10461.457,E2 10461.457} C_VEL
LIN {X 0,Y 405.884,Z 722.892,A -85,B 0,C 180,E1 10462.718,E2 10462.718} C_VEL
LIN {X 0,Y 393.383,Z 685.03,A -85,B 0,C 180,E1 10464.613,E2 10464.613} C_VEL
LIN {X 0,Y 393.135,Z 685.03,A -85,B 0,C 180,E1 10472.496,E2 10472.496} C_VEL
LIN {X 0,Y 393.115,Z 685.03,A -85,B 0,C 180,E1 10479.842,E2 10479.842} C_VEL
LIN {X 0,Y 393.063,Z 685.03,A -85,B 0,C 180,E1 10486.826,E2 10486.826} C_VEL
LIN {X 0,Y 393.062,Z 685.03,A -85,B 0,C 180,E1 10493.712,E2 10493.712} C_VEL
LIN {X 0,Y 393.237,Z 685.434,A -85,B 0,C 180,E1 10497.186,E2 10497.186} C_VEL
LIN {X 0,Y 408.756,Z 722.253,A -85,B 0,C 180,E1 10499.63,E2 10499.63} C_VEL
LIN {X 0,Y 414.148,Z 741.592,A -85,B 0,C 180,E1 10501.057,E2 10501.057} C_VEL
LIN {X 0,Y 411.233,Z 773.106,A -85,B 0,C 180,E1 10503.136,E2 10503.136} C_VEL
LIN {X 0,Y 407.662,Z 801.754,A -85,B 0,C 180,E1 10505.968,E2 10505.968} C_VEL
LIN {X 0,Y 403.646,Z 827.277,A -85,B 0,C 180,E1 10509.591,E2 10509.591} C_VEL
LIN {X 0,Y 400.395,Z 846.783,A -85,B 0,C 180,E1 10513.543,E2 10513.543} C_VEL
LIN {X 0,Y 398.089,Z 861.852,A -85,B 0,C 180,E1 10517.962,E2 10517.962} C_VEL
LIN {X 0,Y 396.755,Z 871.376,A -85,B 0,C 180,E1 10522.346,E2 10522.346} C_VEL
LIN {X 0,Y 396.229,Z 875.598,A -85,B 0,C 180,E1 10525.628,E2 10525.628} C_VEL
LIN {X 0,Y 396.123,Z 877.567,A -85,B 0,C 180,E1 10529.997,E2 10529.997} C_VEL
LIN {X 0,Y 396.378,Z 874.381,A -85,B 0,C 180,E1 10535.458,E2 10535.458} C_VEL
LIN {X 0,Y 397.521,Z 865.891,A -85,B 0,C 180,E1 10540.33,E2 10540.33} C_VEL
LIN {X 0,Y 399.59,Z 851.905,A -85,B 0,C 180,E1 10545.045,E2 10545.045} C_VEL
LIN {X 0,Y 402.921,Z 832.28,A -85,B 0,C 180,E1 10549.411,E2 10549.411} C_VEL
LIN {X 0,Y 406.602,Z 808.693,A -85,B 0,C 180,E1 10553.077,E2 10553.077} C_VEL
LIN {X 0,Y 410.231,Z 781.516,A -85,B 0,C 180,E1 10556.043,E2 10556.043} C_VEL
LIN {X 0,Y 413.374,Z 750.922,A -85,B 0,C 180,E1 10558.329,E2 10558.329} C_VEL
LIN {X 0,Y 413.474,Z 737.506,A -85,B 0,C 180,E1 10559.137,E2 10559.137} C_VEL
LIN {X 0,Y 402.72,Z 706.776,A -85,B 0,C 180,E1 10561.339,E2 10561.339} C_VEL
LIN {X 0,Y 393.238,Z 685.03,A -85,B 0,C 180,E1 10562.823,E2 10562.823} C_VEL
LIN {X 0,Y 393.045,Z 685.03,A -85,B 0,C 180,E1 10569.852,E2 10569.852} C_VEL
LIN {X 0,Y 393.035,Z 685.03,A -85,B 0,C 180,E1 10576.841,E2 10576.841} C_VEL
LIN {X 0,Y 393.056,Z 685.03,A -85,B 0,C 180,E1 10583.727,E2 10583.727} C_VEL
LIN {X 0,Y 393.189,Z 685.03,A -85,B 0,C 180,E1 10590.08,E2 10590.08} C_VEL
LIN {X 0,Y 393.45,Z 685.03,A -85,B 0,C 180,E1 10597.455,E2 10597.455} C_VEL
LIN {X 0,Y 393.845,Z 685.03,A -85,B 0,C 180,E1 10604.449,E2 10604.449} C_VEL
LIN {X 0,Y 394.049,Z 685.03,A -85,B 0,C 180,E1 10611.195,E2 10611.195} C_VEL
LIN {X 0,Y 394.325,Z 685.03,A -85,B 0,C 180,E1 10617.812,E2 10617.812} C_VEL
LIN {X 0,Y 394.223,Z 685.03,A -85,B 0,C 180,E1 10624.395,E2 10624.395} C_VEL
LIN {X 0,Y 393.881,Z 685.03,A -85,B 0,C 180,E1 10631.048,E2 10631.048} C_VEL
LIN {X 0,Y 393.613,Z 685.03,A -85,B 0,C 180,E1 10637.864,E2 10637.864} C_VEL
LIN {X 0,Y 393.32,Z 685.03,A -85,B 0,C 180,E1 10644.965,E2 10644.965} C_VEL
LIN {X 0,Y 393.129,Z 685.03,A -85,B 0,C 180,E1 10652.508,E2 10652.508} C_VEL
LIN {X 0,Y 393.119,Z 685.03,A -85,B 0,C 180,E1 10659.853,E2 10659.853} C_VEL
LIN {X 0,Y 393.095,Z 685.382,A -85,B 0,C 180,E1 10661.644,E2 10661.644} C_VEL
LIN {X 0,Y 403.253,Z 712.594,A -85,B 0,C 180,E1 10664.938,E2 10664.938} C_VEL
LIN {X 0,Y 426.756,Z 764.302,A -85,B 0,C 180,E1 10668.713,E2 10668.713} C_VEL
LIN {X 0,Y 422.445,Z 807.305,A -85,B 0,C 180,E1 10670.404,E2 10670.404} C_VEL
LIN {X 0,Y 416.949,Z 847.871,A -85,B 0,C 180,E1 10672.94,E2 10672.94} C_VEL
LIN {X 0,Y 411.191,Z 884.72,A -85,B 0,C 180,E1 10676.22,E2 10676.22} C_VEL
LIN {X 0,Y 405.754,Z 917.452,A -85,B 0,C 180,E1 10680.173,E2 10680.173} C_VEL
LIN {X 0,Y 401.188,Z 945.582,A -85,B 0,C 180,E1 10684.721,E2 10684.721} C_VEL
LIN {X 0,Y 397.733,Z 969.843,A -85,B 0,C 180,E1 10690.037,E2 10690.037} C_VEL
LIN {X 0,Y 395.865,Z 986.532,A -85,B 0,C 180,E1 10695.092,E2 10695.092} C_VEL
LIN {X 0,Y 395.23,Z 995.373,A -85,B 0,C 180,E1 10698.802,E2 10698.802} C_VEL
LIN {X 0,Y 392.622,Z 998.519,A -85,B 0,C 180,E1 10700.617,E2 10700.617} C_VEL
LIN {X 0,Y 386.988,Z 1002.086,A -85,B 0,C 180,E1 10703.715,E2 10703.715} C_VEL
LIN {X 0,Y 386.933,Z 1005.053,A -85,B 0,C 180,E1 10707.768,E2 10707.768} C_VEL
LIN {X 0,Y 386.982,Z 1004.906,A -85,B 0,C 180,E1 10712.238,E2 10712.238} C_VEL
LIN {X 0,Y 387.159,Z 999.638,A -85,B 0,C 180,E1 10717.844,E2 10717.844} C_VEL
LIN {X 0,Y 387.765,Z 988.738,A -85,B 0,C 180,E1 10723.373,E2 10723.373} C_VEL
LIN {X 0,Y 389.177,Z 972.956,A -85,B 0,C 180,E1 10728.519,E2 10728.519} C_VEL
LIN {X 0,Y 391.863,Z 951.291,A -85,B 0,C 180,E1 10733.553,E2 10733.553} C_VEL
LIN {X 0,Y 395.722,Z 923.748,A -85,B 0,C 180,E1 10738.284,E2 10738.284} C_VEL
LIN {X 0,Y 400.663,Z 889.878,A -85,B 0,C 180,E1 10742.625,E2 10742.625} C_VEL
LIN {X 0,Y 406.39,Z 850.944,A -85,B 0,C 180,E1 10746.314,E2 10746.314} C_VEL
LIN {X 0,Y 412.149,Z 809.07,A -85,B 0,C 180,E1 10749.18,E2 10749.18} C_VEL
LIN {X 0,Y 417.12,Z 764.311,A -85,B 0,C 180,E1 10751.288,E2 10751.288} C_VEL
LIN {X 0,Y 408.555,Z 732.927,A -85,B 0,C 180,E1 10753.898,E2 10753.898} C_VEL
LIN {X 0,Y 402.438,Z 715.23,A -85,B 0,C 180,E1 10755.909,E2 10755.909} C_VEL
LIN {X 0,Y 397.29,Z 704.263,A -85,B 0,C 180,E1 10757.974,E2 10757.974} C_VEL
LIN {X 0,Y 394.231,Z 699.028,A -85,B 0,C 180,E1 10759.645,E2 10759.645} C_VEL
LIN {X 0,Y 391.148,Z 694.64,A -85,B 0,C 180,E1 10763.448,E2 10763.448} C_VEL
LIN {X 0,Y 392.557,Z 697.754,A -85,B 0,C 180,E1 10766.846,E2 10766.846} C_VEL
LIN {X 0,Y 395.596,Z 702.623,A -85,B 0,C 180,E1 10769.074,E2 10769.074} C_VEL
LIN {X 0,Y 400.865,Z 712.782,A -85,B 0,C 180,E1 10771.708,E2 10771.708} C_VEL
LIN {X 0,Y 407.265,Z 729.28,A -85,B 0,C 180,E1 10774.234,E2 10774.234} C_VEL
LIN {X 0,Y 408.304,Z 735.432,A -85,B 0,C 180,E1 10774.8,E2 10774.8} C_VEL
LIN {X 0,Y 403.167,Z 787.888,A -85,B 0,C 180,E1 10777.323,E2 10777.323} C_VEL
LIN {X 0,Y 400.477,Z 814.967,A -85,B 0,C 180,E1 10779.455,E2 10779.455} C_VEL
LIN {X 0,Y 397.344,Z 838.674,A -85,B 0,C 180,E1 10782.309,E2 10782.309} C_VEL
LIN {X 0,Y 394.15,Z 858.415,A -85,B 0,C 180,E1 10785.87,E2 10785.87} C_VEL
LIN {X 0,Y 391.495,Z 872.838,A -85,B 0,C 180,E1 10789.942,E2 10789.942} C_VEL
LIN {X 0,Y 390.161,Z 880.042,A -85,B 0,C 180,E1 10793.333,E2 10793.333} C_VEL
LIN {X 0,Y 389.247,Z 884.09,A -85,B 0,C 180,E1 10797.773,E2 10797.773} C_VEL
LIN {X 0,Y 388.998,Z 882.338,A -85,B 0,C 180,E1 10802.218,E2 10802.218} C_VEL
LIN {X 0,Y 389.248,Z 874.768,A -85,B 0,C 180,E1 10806.673,E2 10806.673} C_VEL
LIN {X 0,Y 390.284,Z 861.992,A -85,B 0,C 180,E1 10810.723,E2 10810.723} C_VEL
LIN {X 0,Y 392.07,Z 843.697,A -85,B 0,C 180,E1 10814.481,E2 10814.481} C_VEL
LIN {X 0,Y 394.325,Z 820.495,A -85,B 0,C 180,E1 10817.695,E2 10817.695} C_VEL
LIN {X 0,Y 396.558,Z 793.125,A -85,B 0,C 180,E1 10820.232,E2 10820.232} C_VEL
LIN {X 0,Y 398.195,Z 763.404,A -85,B 0,C 180,E1 10821.924,E2 10821.924} C_VEL
LIN {X 0,Y 398.73,Z 725.137,A -85,B 0,C 180,E1 10823.084,E2 10823.084} C_VEL
LIN {X 0,Y 385.402,Z 685.03,A -85,B 0,C 180,E1 10825.129,E2 10825.129} C_VEL
LIN {X 0,Y 385.179,Z 685.03,A -85,B 0,C 180,E1 10830.608,E2 10830.608} C_VEL
LIN {X 0,Y 385.154,Z 685.03,A -85,B 0,C 180,E1 10835.983,E2 10835.983} C_VEL
LIN {X 0,Y 385.081,Z 685.03,A -85,B 0,C 180,E1 10841.871,E2 10841.871} C_VEL
LIN {X 0,Y 385.078,Z 685.03,A -85,B 0,C 180,E1 10848.22,E2 10848.22} C_VEL
LIN {X 0,Y 385.177,Z 685.03,A -85,B 0,C 180,E1 10855.341,E2 10855.341} C_VEL
LIN {X 0,Y 385.308,Z 685.03,A -85,B 0,C 180,E1 10856.344,E2 10856.344} C_VEL
LIN {X 0,Y 401.963,Z 724.538,A -85,B 0,C 180,E1 10859.108,E2 10859.108} C_VEL
LIN {X 0,Y 407.206,Z 744.502,A -85,B 0,C 180,E1 10860.614,E2 10860.614} C_VEL
LIN {X 0,Y 404.096,Z 775.946,A -85,B 0,C 180,E1 10862.772,E2 10862.772} C_VEL
LIN {X 0,Y 400.377,Z 804.078,A -85,B 0,C 180,E1 10865.65,E2 10865.65} C_VEL
LIN {X 0,Y 396.439,Z 827.922,A -85,B 0,C 180,E1 10869.099,E2 10869.099} C_VEL
LIN {X 0,Y 392.812,Z 848.613,A -85,B 0,C 180,E1 10873.365,E2 10873.365} C_VEL
LIN {X 0,Y 390.445,Z 863.099,A -85,B 0,C 180,E1 10877.723,E2 10877.723} C_VEL
LIN {X 0,Y 388.983,Z 872.906,A -85,B 0,C 180,E1 10882.371,E2 10882.371} C_VEL
LIN {X 0,Y 388.445,Z 876.845,A -85,B 0,C 180,E1 10885.54,E2 10885.54} C_VEL
LIN {X 0,Y 388.323,Z 878.814,A -85,B 0,C 180,E1 10889.997,E2 10889.997} C_VEL
LIN {X 0,Y 388.447,Z 876.755,A -85,B 0,C 180,E1 10894.453,E2 10894.453} C_VEL
LIN {X 0,Y 389.488,Z 869.446,A -85,B 0,C 180,E1 10899.474,E2 10899.474} C_VEL
LIN {X 0,Y 391.314,Z 857.886,A -85,B 0,C 180,E1 10903.944,E2 10903.944} C_VEL
LIN {X 0,Y 394.311,Z 840.524,A -85,B 0,C 180,E1 10908.402,E2 10908.402} C_VEL
LIN {X 0,Y 397.986,Z 818.687,A -85,B 0,C 180,E1 10912.279,E2 10912.279} C_VEL
LIN {X 0,Y 402.099,Z 791.482,A -85,B 0,C 180,E1 10915.674,E2 10915.674} C_VEL
LIN {X 0,Y 405.696,Z 761.588,A -85,B 0,C 180,E1 10918.232,E2 10918.232} C_VEL
LIN {X 0,Y 406.96,Z 741.113,A -85,B 0,C 180,E1 10919.507,E2 10919.507} C_VEL
LIN {X 0,Y 396.496,Z 710.419,A -85,B 0,C 180,E1 10921.819,E2 10921.819} C_VEL
LIN {X 0,Y 385.289,Z 685.03,A -85,B 0,C 180,E1 10923.586,E2 10923.586} C_VEL
LIN {X 0,Y 385.112,Z 685.03,A -85,B 0,C 180,E1 10928.822,E2 10928.822} C_VEL
LIN {X 0,Y 385.026,Z 685.03,A -85,B 0,C 180,E1 10935.145,E2 10935.145} C_VEL
LIN {X 0,Y 385.16,Z 685.03,A -85,B 0,C 180,E1 10941.587,E2 10941.587} C_VEL
LIN {X 0,Y 385.12,Z 685.03,A -85,B 0,C 180,E1 10946.741,E2 10946.741} C_VEL
LIN {X 0,Y 385.31,Z 685.03,A -85,B 0,C 180,E1 10951.977,E2 10951.977} C_VEL
LIN {X 0,Y 385.607,Z 685.03,A -85,B 0,C 180,E1 10959.385,E2 10959.385} C_VEL
LIN {X 0,Y 386.014,Z 685.03,A -85,B 0,C 180,E1 10966.441,E2 10966.441} C_VEL
LIN {X 0,Y 386.239,Z 685.03,A -85,B 0,C 180,E1 10973.275,E2 10973.275} C_VEL
LIN {X 0,Y 386.574,Z 685.03,A -85,B 0,C 180,E1 10980.005,E2 10980.005} C_VEL
LIN {X 0,Y 386.234,Z 685.03,A -85,B 0,C 180,E1 10986.735,E2 10986.735} C_VEL
LIN {X 0,Y 385.86,Z 685.03,A -85,B 0,C 180,E1 10993.575,E2 10993.575} C_VEL
LIN {X 0,Y 385.571,Z 685.03,A -85,B 0,C 180,E1 11000.627,E2 11000.627} C_VEL
LIN {X 0,Y 385.25,Z 685.03,A -85,B 0,C 180,E1 11008.039,E2 11008.039} C_VEL
LIN {X 0,Y 385.151,Z 685.03,A -85,B 0,C 180,E1 11015.996,E2 11015.996} C_VEL
LIN {X 0,Y 385.193,Z 685.423,A -85,B 0,C 180,E1 11020.764,E2 11020.764} C_VEL
LIN {X 0,Y 394.784,Z 711.159,A -85,B 0,C 180,E1 11023.997,E2 11023.997} C_VEL
LIN {X 0,Y 417.192,Z 760.721,A -85,B 0,C 180,E1 11027.713,E2 11027.713} C_VEL
LIN {X 0,Y 419.909,Z 768.916,A -85,B 0,C 180,E1 11028.268,E2 11028.268} C_VEL
LIN {X 0,Y 415.201,Z 810.466,A -85,B 0,C 180,E1 11030.021,E2 11030.021} C_VEL
LIN {X 0,Y 409.591,Z 849.767,A -85,B 0,C 180,E1 11032.587,E2 11032.587} C_VEL
LIN {X 0,Y 403.882,Z 884.75,A -85,B 0,C 180,E1 11035.789,E2 11035.789} C_VEL
LIN {X 0,Y 398.155,Z 917.693,A -85,B 0,C 180,E1 11039.858,E2 11039.858} C_VEL
LIN {X 0,Y 393.465,Z 945.494,A -85,B 0,C 180,E1 11044.476,E2 11044.476} C_VEL
LIN {X 0,Y 389.992,Z 968.543,A -85,B 0,C 180,E1 11049.623,E2 11049.623} C_VEL
LIN {X 0,Y 388.047,Z 985.342,A -85,B 0,C 180,E1 11054.785,E2 11054.785} C_VEL
LIN {X 0,Y 387.286,Z 996.74,A -85,B 0,C 180,E1 11059.905,E2 11059.905} C_VEL
LIN {X 0,Y 386.988,Z 1002.086,A -85,B 0,C 180,E1 11063.715,E2 11063.715} C_VEL
LIN {X 0,Y 384.382,Z 1003.521,A -85,B 0,C 180,E1 11065.609,E2 11065.609} C_VEL
LIN {X 0,Y 379.052,Z 1004.138,A -85,B 0,C 180,E1 11068.813,E2 11068.813} C_VEL
LIN {X 0,Y 379.155,Z 1003.779,A -85,B 0,C 180,E1 11072.285,E2 11072.285} C_VEL
LIN {X 0,Y 379.284,Z 999.958,A -85,B 0,C 180,E1 11076.859,E2 11076.859} C_VEL
LIN {X 0,Y 379.768,Z 990.199,A -85,B 0,C 180,E1 11082.451,E2 11082.451} C_VEL
LIN {X 0,Y 381.061,Z 975.635,A -85,B 0,C 180,E1 11087.68,E2 11087.68} C_VEL
LIN {X 0,Y 383.676,Z 953.691,A -85,B 0,C 180,E1 11093.165,E2 11093.165} C_VEL
LIN {X 0,Y 387.556,Z 926.884,A -85,B 0,C 180,E1 11098.058,E2 11098.058} C_VEL
LIN {X 0,Y 392.678,Z 893.891,A -85,B 0,C 180,E1 11102.553,E2 11102.553} C_VEL
LIN {X 0,Y 398.659,Z 855.614,A -85,B 0,C 180,E1 11106.434,E2 11106.434} C_VEL
LIN {X 0,Y 404.865,Z 813.541,A -85,B 0,C 180,E1 11109.526,E2 11109.526} C_VEL
LIN {X 0,Y 410.737,Z 771.014,A -85,B 0,C 180,E1 11111.669,E2 11111.669} C_VEL
LIN {X 0,Y 410.072,Z 765.039,A -85,B 0,C 180,E1 11112.084,E2 11112.084} C_VEL
LIN {X 0,Y 401.018,Z 727.769,A -85,B 0,C 180,E1 11115.515,E2 11115.515} C_VEL
LIN {X 0,Y 395.335,Z 713.147,A -85,B 0,C 180,E1 11117.867,E2 11117.867} C_VEL
LIN {X 0,Y 391.76,Z 706.382,A -85,B 0,C 180,E1 11119.886,E2 11119.886} C_VEL
LIN {X 0,Y 389.14,Z 702.703,A -85,B 0,C 180,E1 11122.582,E2 11122.582} C_VEL
LIN {X 0,Y 388.851,Z 702.697,A -85,B 0,C 180,E1 11124.591,E2 11124.591} C_VEL
LIN {X 0,Y 391.42,Z 707.187,A -85,B 0,C 180,E1 11128.022,E2 11128.022} C_VEL
LIN {X 0,Y 396.372,Z 717.978,A -85,B 0,C 180,E1 11131.131,E2 11131.131} C_VEL
LIN {X 0,Y 402.003,Z 733.826,A -85,B 0,C 180,E1 11133.706,E2 11133.706} C_VEL
LIN {X 0,Y 402.34,Z 739.004,A -85,B 0,C 180,E1 11134.141,E2 11134.141} C_VEL
LIN {X 0,Y 396.652,Z 790.07,A -85,B 0,C 180,E1 11136.757,E2 11136.757} C_VEL
LIN {X 0,Y 393.708,Z 816.846,A -85,B 0,C 180,E1 11138.938,E2 11138.938} C_VEL
LIN {X 0,Y 390.407,Z 839.727,A -85,B 0,C 180,E1 11141.747,E2 11141.747} C_VEL
LIN {X 0,Y 387.017,Z 859.247,A -85,B 0,C 180,E1 11145.315,E2 11145.315} C_VEL
LIN {X 0,Y 384.148,Z 873.623,A -85,B 0,C 180,E1 11149.367,E2 11149.367} C_VEL
LIN {X 0,Y 382.493,Z 881.68,A -85,B 0,C 180,E1 11153.198,E2 11153.198} C_VEL
LIN {X 0,Y 381.492,Z 885.557,A -85,B 0,C 180,E1 11157.728,E2 11157.728} C_VEL
LIN {X 0,Y 381.23,Z 883.625,A -85,B 0,C 180,E1 11162.263,E2 11162.263} C_VEL
LIN {X 0,Y 381.498,Z 875.901,A -85,B 0,C 180,E1 11166.809,E2 11166.809} C_VEL
LIN {X 0,Y 382.625,Z 862.404,A -85,B 0,C 180,E1 11171.079,E2 11171.079} C_VEL
LIN {X 0,Y 384.454,Z 844.468,A -85,B 0,C 180,E1 11174.775,E2 11174.775} C_VEL
LIN {X 0,Y 386.782,Z 821.518,A -85,B 0,C 180,E1 11177.991,E2 11177.991} C_VEL
LIN {X 0,Y 389.024,Z 794.804,A -85,B 0,C 180,E1 11180.523,E2 11180.523} C_VEL
LIN {X 0,Y 390.772,Z 765.715,A -85,B 0,C 180,E1 11182.248,E2 11182.248} C_VEL
LIN {X 0,Y 391.338,Z 726.459,A -85,B 0,C 180,E1 11183.5,E2 11183.5} C_VEL
LIN {X 0,Y 377.429,Z 685.03,A -85,B 0,C 180,E1 11185.73,E2 11185.73} C_VEL
LIN {X 0,Y 377.179,Z 685.03,A -85,B 0,C 180,E1 11192.832,E2 11192.832} C_VEL
LIN {X 0,Y 377.131,Z 685.03,A -85,B 0,C 180,E1 11199.796,E2 11199.796} C_VEL
LIN {X 0,Y 377.074,Z 685.03,A -85,B 0,C 180,E1 11207.124,E2 11207.124} C_VEL
LIN {X 0,Y 377.239,Z 685.03,A -85,B 0,C 180,E1 11214.447,E2 11214.447} C_VEL
LIN {X 0,Y 377.289,Z 685.03,A -85,B 0,C 180,E1 11215.511,E2 11215.511} C_VEL
LIN {X 0,Y 394.569,Z 725.004,A -85,B 0,C 180,E1 11218.427,E2 11218.427} C_VEL
LIN {X 0,Y 400.342,Z 746.945,A -85,B 0,C 180,E1 11220.133,E2 11220.133} C_VEL
LIN {X 0,Y 397.03,Z 778.777,A -85,B 0,C 180,E1 11222.4,E2 11222.4} C_VEL
LIN {X 0,Y 393.099,Z 806.403,A -85,B 0,C 180,E1 11225.321,E2 11225.321} C_VEL
LIN {X 0,Y 388.925,Z 830.621,A -85,B 0,C 180,E1 11228.943,E2 11228.943} C_VEL
LIN {X 0,Y 385.137,Z 850.908,A -85,B 0,C 180,E1 11233.297,E2 11233.297} C_VEL
LIN {X 0,Y 382.558,Z 865.77,A -85,B 0,C 180,E1 11238.044,E2 11238.044} C_VEL
LIN {X 0,Y 381.084,Z 875.544,A -85,B 0,C 180,E1 11243.174,E2 11243.174} C_VEL
LIN {X 0,Y 380.582,Z 879.537,A -85,B 0,C 180,E1 11247.724,E2 11247.724} C_VEL
LIN {X 0,Y 380.582,Z 879.5,A -85,B 0,C 180,E1 11252.269,E2 11252.269} C_VEL
LIN {X 0,Y 381.104,Z 875.429,A -85,B 0,C 180,E1 11256.819,E2 11256.819} C_VEL
LIN {X 0,Y 382.575,Z 865.55,A -85,B 0,C 180,E1 11261.948,E2 11261.948} C_VEL
LIN {X 0,Y 385.248,Z 850.395,A -85,B 0,C 180,E1 11266.732,E2 11266.732} C_VEL
LIN {X 0,Y 389.044,Z 829.816,A -85,B 0,C 180,E1 11271.1,E2 11271.1} C_VEL
LIN {X 0,Y 393.341,Z 804.652,A -85,B 0,C 180,E1 11274.807,E2 11274.807} C_VEL
LIN {X 0,Y 397.294,Z 776.187,A -85,B 0,C 180,E1 11277.726,E2 11277.726} C_VEL
LIN {X 0,Y 400.368,Z 744.337,A -85,B 0,C 180,E1 11279.92,E2 11279.92} C_VEL
LIN {X 0,Y 390.306,Z 714.045,A -85,B 0,C 180,E1 11282.308,E2 11282.308} C_VEL
LIN {X 0,Y 377.286,Z 685.03,A -85,B 0,C 180,E1 11284.407,E2 11284.407} C_VEL
LIN {X 0,Y 377.055,Z 685.03,A -85,B 0,C 180,E1 11290.515,E2 11290.515} C_VEL
LIN {X 0,Y 377.045,Z 685.03,A -85,B 0,C 180,E1 11297.139,E2 11297.139} C_VEL
LIN {X 0,Y 377.18,Z 685.03,A -85,B 0,C 180,E1 11303.143,E2 11303.143} C_VEL
LIN {X 0,Y 377.211,Z 685.03,A -85,B 0,C 180,E1 11308.673,E2 11308.673} C_VEL
LIN {X 0,Y 377.407,Z 685.03,A -85,B 0,C 180,E1 11313.916,E2 11313.916} C_VEL
LIN {X 0,Y 377.789,Z 685.03,A -85,B 0,C 180,E1 11321.372,E2 11321.372} C_VEL
LIN {X 0,Y 378.165,Z 685.03,A -85,B 0,C 180,E1 11328.498,E2 11328.498} C_VEL
LIN {X 0,Y 378.449,Z 685.03,A -85,B 0,C 180,E1 11335.432,E2 11335.432} C_VEL
LIN {X 0,Y 378.653,Z 685.03,A -85,B 0,C 180,E1 11342.289,E2 11342.289} C_VEL
LIN {X 0,Y 378.115,Z 685.03,A -85,B 0,C 180,E1 11349.19,E2 11349.19} C_VEL
LIN {X 0,Y 377.778,Z 685.03,A -85,B 0,C 180,E1 11356.535,E2 11356.535} C_VEL
LIN {X 0,Y 377.503,Z 685.03,A -85,B 0,C 180,E1 11363.565,E2 11363.565} C_VEL
LIN {X 0,Y 377.266,Z 685.03,A -85,B 0,C 180,E1 11368.687,E2 11368.687} C_VEL
LIN {X 0,Y 377.181,Z 685.03,A -85,B 0,C 180,E1 11374.066,E2 11374.066} C_VEL
LIN {X 0,Y 377.332,Z 685.355,A -85,B 0,C 180,E1 11379.869,E2 11379.869} C_VEL
LIN {X 0,Y 386.798,Z 710.854,A -85,B 0,C 180,E1 11383.103,E2 11383.103} C_VEL
LIN {X 0,Y 408.652,Z 758.661,A -85,B 0,C 180,E1 11386.829,E2 11386.829} C_VEL
LIN {X 0,Y 413.156,Z 771.005,A -85,B 0,C 180,E1 11387.747,E2 11387.747} C_VEL
LIN {X 0,Y 408.279,Z 811.237,A -85,B 0,C 180,E1 11389.503,E2 11389.503} C_VEL
LIN {X 0,Y 402.57,Z 849.555,A -85,B 0,C 180,E1 11392.059,E2 11392.059} C_VEL
LIN {X 0,Y 396.566,Z 884.87,A -85,B 0,C 180,E1 11395.363,E2 11395.363} C_VEL
LIN {X 0,Y 390.877,Z 916.022,A -85,B 0,C 180,E1 11399.261,E2 11399.261} C_VEL
LIN {X 0,Y 385.817,Z 944.778,A -85,B 0,C 180,E1 11404.103,E2 11404.103} C_VEL
LIN {X 0,Y 382.148,Z 968.307,A -85,B 0,C 180,E1 11409.488,E2 11409.488} C_VEL
LIN {X 0,Y 380.104,Z 985.655,A -85,B 0,C 180,E1 11415.049,E2 11415.049} C_VEL
LIN {X 0,Y 379.302,Z 997.493,A -85,B 0,C 180,E1 11420.846,E2 11420.846} C_VEL
LIN {X 0,Y 379.129,Z 1002.706,A -85,B 0,C 180,E1 11425.437,E2 11425.437} C_VEL
LIN {X 0,Y 379.052,Z 1004.138,A -85,B 0,C 180,E1 11428.813,E2 11428.813} C_VEL
LIN {X 0,Y 376.561,Z 1003.89,A -85,B 0,C 180,E1 11430.765,E2 11430.765} C_VEL
LIN {X 0,Y 371.353,Z 1001.906,A -85,B 0,C 180,E1 11433.699,E2 11433.699} C_VEL
LIN {X 0,Y 371.285,Z 1001.563,A -85,B 0,C 180,E1 11434.039,E2 11434.039} C_VEL
LIN {X 0,Y 371.577,Z 995.383,A -85,B 0,C 180,E1 11439.353,E2 11439.353} C_VEL
LIN {X 0,Y 372.25,Z 984.078,A -85,B 0,C 180,E1 11444.681,E2 11444.681} C_VEL
LIN {X 0,Y 374.053,Z 967.024,A -85,B 0,C 180,E1 11450.059,E2 11450.059} C_VEL
LIN {X 0,Y 377.351,Z 943.057,A -85,B 0,C 180,E1 11455.466,E2 11455.466} C_VEL
LIN {X 0,Y 382.109,Z 912.999,A -85,B 0,C 180,E1 11460.449,E2 11460.449} C_VEL
LIN {X 0,Y 387.768,Z 878.382,A -85,B 0,C 180,E1 11464.737,E2 11464.737} C_VEL
LIN {X 0,Y 394.423,Z 837.789,A -85,B 0,C 180,E1 11468.462,E2 11468.462} C_VEL
LIN {X 0,Y 401.265,Z 794.247,A -85,B 0,C 180,E1 11471.311,E2 11471.311} C_VEL
LIN {X 0,Y 404.421,Z 769.511,A -85,B 0,C 180,E1 11472.54,E2 11472.54} C_VEL
LIN {X 0,Y 396.572,Z 732.686,A -85,B 0,C 180,E1 11476.136,E2 11476.136} C_VEL
LIN {X 0,Y 391.783,Z 718.619,A -85,B 0,C 180,E1 11478.532,E2 11478.532} C_VEL
LIN {X 0,Y 388.866,Z 713.39,A -85,B 0,C 180,E1 11480.356,E2 11480.356} C_VEL
LIN {X 0,Y 386.392,Z 710.045,A -85,B 0,C 180,E1 11484.138,E2 11484.138} C_VEL
LIN {X 0,Y 388.283,Z 714.176,A -85,B 0,C 180,E1 11487.732,E2 11487.732} C_VEL
LIN {X 0,Y 392.113,Z 723.522,A -85,B 0,C 180,E1 11490.585,E2 11490.585} C_VEL
LIN {X 0,Y 396.642,Z 737.509,A -85,B 0,C 180,E1 11493.035,E2 11493.035} C_VEL
LIN {X 0,Y 396.576,Z 742.56,A -85,B 0,C 180,E1 11493.44,E2 11493.44} C_VEL
LIN {X 0,Y 390.154,Z 793.428,A -85,B 0,C 180,E1 11496.234,E2 11496.234} C_VEL
LIN {X 0,Y 386.638,Z 821.482,A -85,B 0,C 180,E1 11498.684,E2 11498.684} C_VEL
LIN {X 0,Y 383.048,Z 843.739,A -85,B 0,C 180,E1 11501.626,E2 11501.626} C_VEL
LIN {X 0,Y 379.413,Z 862.626,A -85,B 0,C 180,E1 11505.309,E2 11505.309} C_VEL
LIN {X 0,Y 376.384,Z 876.534,A -85,B 0,C 180,E1 11509.549,E2 11509.549} C_VEL
LIN {X 0,Y 374.489,Z 884.795,A -85,B 0,C 180,E1 11514.214,E2 11514.214} C_VEL
LIN {X 0,Y 373.756,Z 887.022,A -85,B 0,C 180,E1 11517.681,E2 11517.681} C_VEL
LIN {X 0,Y 373.438,Z 884.916,A -85,B 0,C 180,E1 11522.31,E2 11522.31} C_VEL
LIN {X 0,Y 373.727,Z 877,A -85,B 0,C 180,E1 11526.952,E2 11526.952} C_VEL
LIN {X 0,Y 374.93,Z 863.328,A -85,B 0,C 180,E1 11531.309,E2 11531.309} C_VEL
LIN {X 0,Y 376.839,Z 845.224,A -85,B 0,C 180,E1 11535.08,E2 11535.08} C_VEL
LIN {X 0,Y 379.304,Z 821.689,A -85,B 0,C 180,E1 11538.401,E2 11538.401} C_VEL
LIN {X 0,Y 381.693,Z 794.238,A -85,B 0,C 180,E1 11540.998,E2 11540.998} C_VEL
LIN {X 0,Y 383.485,Z 764.228,A -85,B 0,C 180,E1 11542.748,E2 11542.748} C_VEL
LIN {X 0,Y 383.877,Z 727.725,A -85,B 0,C 180,E1 11543.928,E2 11543.928} C_VEL
LIN {X 0,Y 369.447,Z 685.03,A -85,B 0,C 180,E1 11546.312,E2 11546.312} C_VEL
LIN {X 0,Y 369.249,Z 685.03,A -85,B 0,C 180,E1 11552.082,E2 11552.082} C_VEL
LIN {X 0,Y 369.157,Z 685.03,A -85,B 0,C 180,E1 11559.035,E2 11559.035} C_VEL
LIN {X 0,Y 369.167,Z 685.03,A -85,B 0,C 180,E1 11565.974,E2 11565.974} C_VEL
LIN {X 0,Y 369.286,Z 685.03,A -85,B 0,C 180,E1 11573.542,E2 11573.542} C_VEL
LIN {X 0,Y 369.37,Z 685.03,A -85,B 0,C 180,E1 11574.612,E2 11574.612} C_VEL
LIN {X 0,Y 387.579,Z 726.539,A -85,B 0,C 180,E1 11577.803,E2 11577.803} C_VEL
LIN {X 0,Y 393.506,Z 749.021,A -85,B 0,C 180,E1 11579.616,E2 11579.616} C_VEL
LIN {X 0,Y 390.123,Z 780.107,A -85,B 0,C 180,E1 11581.879,E2 11581.879} C_VEL
LIN {X 0,Y 385.844,Z 808.727,A -85,B 0,C 180,E1 11584.979,E2 11584.979} C_VEL
LIN {X 0,Y 381.44,Z 832.902,A -85,B 0,C 180,E1 11588.719,E2 11588.719} C_VEL
LIN {X 0,Y 377.514,Z 852.906,A -85,B 0,C 180,E1 11593.15,E2 11593.15} C_VEL
LIN {X 0,Y 374.913,Z 867.017,A -85,B 0,C 180,E1 11597.797,E2 11597.797} C_VEL
LIN {X 0,Y 373.34,Z 876.79,A -85,B 0,C 180,E1 11603.031,E2 11603.031} C_VEL
LIN {X 0,Y 372.806,Z 880.782,A -85,B 0,C 180,E1 11607.677,E2 11607.677} C_VEL
LIN {X 0,Y 372.805,Z 880.744,A -85,B 0,C 180,E1 11612.316,E2 11612.316} C_VEL
LIN {X 0,Y 373.358,Z 876.677,A -85,B 0,C 180,E1 11616.961,E2 11616.961} C_VEL
LIN {X 0,Y 374.932,Z 866.8,A -85,B 0,C 180,E1 11622.196,E2 11622.196} C_VEL
LIN {X 0,Y 377.806,Z 851.428,A -85,B 0,C 180,E1 11627.129,E2 11627.129} C_VEL
LIN {X 0,Y 381.789,Z 831.058,A -85,B 0,C 180,E1 11631.521,E2 11631.521} C_VEL
LIN {X 0,Y 386.293,Z 805.889,A -85,B 0,C 180,E1 11635.291,E2 11635.291} C_VEL
LIN {X 0,Y 390.366,Z 777.724,A -85,B 0,C 180,E1 11638.232,E2 11638.232} C_VEL
LIN {X 0,Y 393.257,Z 745.593,A -85,B 0,C 180,E1 11640.52,E2 11640.52} C_VEL
LIN {X 0,Y 383.603,Z 716.404,A -85,B 0,C 180,E1 11642.9,E2 11642.9} C_VEL
LIN {X 0,Y 369.349,Z 685.03,A -85,B 0,C 180,E1 11645.291,E2 11645.291} C_VEL
LIN {X 0,Y 369.108,Z 685.03,A -85,B 0,C 180,E1 11652.631,E2 11652.631} C_VEL
LIN {X 0,Y 369.151,Z 685.03,A -85,B 0,C 180,E1 11659.164,E2 11659.164} C_VEL
LIN {X 0,Y 369.19,Z 685.03,A -85,B 0,C 180,E1 11665.104,E2 11665.104} C_VEL
LIN {X 0,Y 369.323,Z 685.03,A -85,B 0,C 180,E1 11670.648,E2 11670.648} C_VEL
LIN {X 0,Y 369.537,Z 685.03,A -85,B 0,C 180,E1 11675.907,E2 11675.907} C_VEL
LIN {X 0,Y 369.985,Z 685.03,A -85,B 0,C 180,E1 11683.418,E2 11683.418} C_VEL
LIN {X 0,Y 370.266,Z 685.03,A -85,B 0,C 180,E1 11690.624,E2 11690.624} C_VEL
LIN {X 0,Y 370.626,Z 685.03,A -85,B 0,C 180,E1 11697.672,E2 11697.672} C_VEL
LIN {X 0,Y 370.749,Z 685.03,A -85,B 0,C 180,E1 11702.338,E2 11702.338} C_VEL
LIN {X 0,Y 370.184,Z 685.03,A -85,B 0,C 180,E1 11709.389,E2 11709.389} C_VEL
LIN {X 0,Y 369.878,Z 685.03,A -85,B 0,C 180,E1 11716.598,E2 11716.598} C_VEL
LIN {X 0,Y 369.511,Z 685.03,A -85,B 0,C 180,E1 11724.106,E2 11724.106} C_VEL
LIN {X 0,Y 369.245,Z 685.03,A -85,B 0,C 180,E1 11732.095,E2 11732.095} C_VEL
LIN {X 0,Y 369.296,Z 685.401,A -85,B 0,C 180,E1 11738.929,E2 11738.929} C_VEL
LIN {X 0,Y 378.359,Z 709.567,A -85,B 0,C 180,E1 11742.111,E2 11742.111} C_VEL
LIN {X 0,Y 400.608,Z 757.66,A -85,B 0,C 180,E1 11746.011,E2 11746.011} C_VEL
LIN {X 0,Y 406.306,Z 773.437,A -85,B 0,C 180,E1 11747.217,E2 11747.217} C_VEL
LIN {X 0,Y 401.115,Z 814.103,A -85,B 0,C 180,E1 11749.093,E2 11749.093} C_VEL
LIN {X 0,Y 394.631,Z 854.799,A -85,B 0,C 180,E1 11751.968,E2 11751.968} C_VEL
LIN {X 0,Y 387.993,Z 891.604,A -85,B 0,C 180,E1 11755.673,E2 11755.673} C_VEL
LIN {X 0,Y 381.968,Z 923.628,A -85,B 0,C 180,E1 11760.085,E2 11760.085} C_VEL
LIN {X 0,Y 377.016,Z 950.901,A -85,B 0,C 180,E1 11765.151,E2 11765.151} C_VEL
LIN {X 0,Y 373.731,Z 972.212,A -85,B 0,C 180,E1 11770.545,E2 11770.545} C_VEL
LIN {X 0,Y 371.924,Z 988.717,A -85,B 0,C 180,E1 11776.518,E2 11776.518} C_VEL
LIN {X 0,Y 371.38,Z 998.035,A -85,B 0,C 180,E1 11781.827,E2 11781.827} C_VEL
LIN {X 0,Y 371.286,Z 1001.618,A -85,B 0,C 180,E1 11785.341,E2 11785.341} C_VEL
LIN {X 0,Y 371.348,Z 1003.229,A -85,B 0,C 180,E1 11790.004,E2 11790.004} C_VEL
LIN {X 0,Y 371.285,Z 1001.563,A -85,B 0,C 180,E1 11794.039,E2 11794.039} C_VEL
LIN {X 0,Y 368.891,Z 999.562,A -85,B 0,C 180,E1 11796.012,E2 11796.012} C_VEL
LIN {X 0,Y 363.764,Z 995.101,A -85,B 0,C 180,E1 11798.947,E2 11798.947} C_VEL
LIN {X 0,Y 363.703,Z 994.533,A -85,B 0,C 180,E1 11799.286,E2 11799.286} C_VEL
LIN {X 0,Y 364.452,Z 982.668,A -85,B 0,C 180,E1 11805.002,E2 11805.002} C_VEL
LIN {X 0,Y 366.347,Z 965.428,A -85,B 0,C 180,E1 11810.5,E2 11810.5} C_VEL
LIN {X 0,Y 369.913,Z 941.027,A -85,B 0,C 180,E1 11816.065,E2 11816.065} C_VEL
LIN {X 0,Y 374.934,Z 910.778,A -85,B 0,C 180,E1 11821.133,E2 11821.133} C_VEL
LIN {X 0,Y 381.149,Z 875.066,A -85,B 0,C 180,E1 11825.599,E2 11825.599} C_VEL
LIN {X 0,Y 388.405,Z 834.125,A -85,B 0,C 180,E1 11829.375,E2 11829.375} C_VEL
LIN {X 0,Y 396.016,Z 789.135,A -85,B 0,C 180,E1 11832.316,E2 11832.316} C_VEL
LIN {X 0,Y 398.479,Z 772.752,A -85,B 0,C 180,E1 11833.148,E2 11833.148} C_VEL
LIN {X 0,Y 392.071,Z 736.912,A -85,B 0,C 180,E1 11836.863,E2 11836.863} C_VEL
LIN {X 0,Y 388.257,Z 724.724,A -85,B 0,C 180,E1 11839.133,E2 11839.133} C_VEL
LIN {X 0,Y 385.886,Z 720.333,A -85,B 0,C 180,E1 11840.836,E2 11840.836} C_VEL
LIN {X 0,Y 383.866,Z 717.697,A -85,B 0,C 180,E1 11843.865,E2 11843.865} C_VEL
LIN {X 0,Y 385.008,Z 720.925,A -85,B 0,C 180,E1 11847.295,E2 11847.295} C_VEL
LIN {X 0,Y 388.173,Z 729.814,A -85,B 0,C 180,E1 11850.186,E2 11850.186} C_VEL
LIN {X 0,Y 391.685,Z 742.194,A -85,B 0,C 180,E1 11852.461,E2 11852.461} C_VEL
LIN {X 0,Y 383.851,Z 795.961,A -85,B 0,C 180,E1 11855.617,E2 11855.617} C_VEL
LIN {X 0,Y 379.985,Z 823.608,A -85,B 0,C 180,E1 11858.139,E2 11858.139} C_VEL
LIN {X 0,Y 375.947,Z 846.384,A -85,B 0,C 180,E1 11861.266,E2 11861.266} C_VEL
LIN {X 0,Y 372.09,Z 864.794,A -85,B 0,C 180,E1 11865.013,E2 11865.013} C_VEL
LIN {X 0,Y 368.874,Z 878.318,A -85,B 0,C 180,E1 11869.301,E2 11869.301} C_VEL
LIN {X 0,Y 366.798,Z 886.424,A -85,B 0,C 180,E1 11874.092,E2 11874.092} C_VEL
LIN {X 0,Y 366.002,Z 888.494,A -85,B 0,C 180,E1 11877.632,E2 11877.632} C_VEL
LIN {X 0,Y 365.67,Z 886.2,A -85,B 0,C 180,E1 11882.36,E2 11882.36} C_VEL
LIN {X 0,Y 365.981,Z 878.082,A -85,B 0,C 180,E1 11887.099,E2 11887.099} C_VEL
LIN {X 0,Y 367.249,Z 864.215,A -85,B 0,C 180,E1 11891.549,E2 11891.549} C_VEL
LIN {X 0,Y 369.236,Z 846.037,A -85,B 0,C 180,E1 11895.369,E2 11895.369} C_VEL
LIN {X 0,Y 371.804,Z 822.11,A -85,B 0,C 180,E1 11898.786,E2 11898.786} C_VEL
LIN {X 0,Y 374.247,Z 795.216,A -85,B 0,C 180,E1 11901.366,E2 11901.366} C_VEL
LIN {X 0,Y 376.126,Z 765.187,A -85,B 0,C 180,E1 11903.158,E2 11903.158} C_VEL
LIN {X 0,Y 376.622,Z 729.59,A -85,B 0,C 180,E1 11904.343,E2 11904.343} C_VEL
LIN {X 0,Y 361.462,Z 685.03,A -85,B 0,C 180,E1 11906.946,E2 11906.946} C_VEL
LIN {X 0,Y 361.22,Z 685.03,A -85,B 0,C 180,E1 11913.321,E2 11913.321} C_VEL
LIN {X 0,Y 361.249,Z 685.03,A -85,B 0,C 180,E1 11918.787,E2 11918.787} C_VEL
LIN {X 0,Y 361.244,Z 685.03,A -85,B 0,C 180,E1 11925.233,E2 11925.233} C_VEL
LIN {X 0,Y 361.271,Z 685.03,A -85,B 0,C 180,E1 11932.51,E2 11932.51} C_VEL
LIN {X 0,Y 361.425,Z 685.03,A -85,B 0,C 180,E1 11933.711,E2 11933.711} C_VEL
LIN {X 0,Y 368.229,Z 699.682,A -85,B 0,C 180,E1 11934.879,E2 11934.879} C_VEL
LIN {X 0,Y 381.381,Z 730.322,A -85,B 0,C 180,E1 11937.338,E2 11937.338} C_VEL
LIN {X 0,Y 386.697,Z 751.161,A -85,B 0,C 180,E1 11939.088,E2 11939.088} C_VEL
LIN {X 0,Y 383.079,Z 782.837,A -85,B 0,C 180,E1 11941.464,E2 11941.464} C_VEL
LIN {X 0,Y 378.572,Z 811.056,A -85,B 0,C 180,E1 11944.622,E2 11944.622} C_VEL
LIN {X 0,Y 373.973,Z 835.08,A -85,B 0,C 180,E1 11948.466,E2 11948.466} C_VEL
LIN {X 0,Y 369.827,Z 855.183,A -85,B 0,C 180,E1 11953.094,E2 11953.094} C_VEL
LIN {X 0,Y 367.024,Z 869.689,A -85,B 0,C 180,E1 11958.133,E2 11958.133} C_VEL
LIN {X 0,Y 365.601,Z 878.036,A -85,B 0,C 180,E1 11962.883,E2 11962.883} C_VEL
LIN {X 0,Y 365.018,Z 882.028,A -85,B 0,C 180,E1 11967.627,E2 11967.627} C_VEL
LIN {X 0,Y 365.017,Z 881.991,A -85,B 0,C 180,E1 11972.366,E2 11972.366} C_VEL
LIN {X 0,Y 365.619,Z 877.924,A -85,B 0,C 180,E1 11977.109,E2 11977.109} C_VEL
LIN {X 0,Y 367.308,Z 868.048,A -85,B 0,C 180,E1 11982.453,E2 11982.453} C_VEL
LIN {X 0,Y 370.346,Z 852.676,A -85,B 0,C 180,E1 11987.485,E2 11987.485} C_VEL
LIN {X 0,Y 374.383,Z 833.093,A -85,B 0,C 180,E1 11991.816,E2 11991.816} C_VEL
LIN {X 0,Y 379.072,Z 808.219,A -85,B 0,C 180,E1 11995.65,E2 11995.65} C_VEL
LIN {X 0,Y 383.31,Z 780.279,A -85,B 0,C 180,E1 11998.67,E2 11998.67} C_VEL
LIN {X 0,Y 386.558,Z 748.182,A -85,B 0,C 180,E1 12001.021,E2 12001.021} C_VEL
LIN {X 0,Y 377.047,Z 718.966,A -85,B 0,C 180,E1 12003.495,E2 12003.495} C_VEL
LIN {X 0,Y 361.384,Z 685.03,A -85,B 0,C 180,E1 12006.21,E2 12006.21} C_VEL
LIN {X 0,Y 361.185,Z 685.03,A -85,B 0,C 180,E1 12011.947,E2 12011.947} C_VEL
LIN {X 0,Y 361.229,Z 685.03,A -85,B 0,C 180,E1 12018.756,E2 12018.756} C_VEL
LIN {X 0,Y 361.2,Z 685.03,A -85,B 0,C 180,E1 12024.215,E2 12024.215} C_VEL
LIN {X 0,Y 361.383,Z 685.03,A -85,B 0,C 180,E1 12031.266,E2 12031.266} C_VEL
LIN {X 0,Y 361.702,Z 685.03,A -85,B 0,C 180,E1 12037.954,E2 12037.954} C_VEL
LIN {X 0,Y 362.177,Z 685.03,A -85,B 0,C 180,E1 12045.53,E2 12045.53} C_VEL
LIN {X 0,Y 362.478,Z 685.03,A -85,B 0,C 180,E1 12052.832,E2 12052.832} C_VEL
LIN {X 0,Y 362.889,Z 685.03,A -85,B 0,C 180,E1 12060.005,E2 12060.005} C_VEL
LIN {X 0,Y 362.461,Z 685.03,A -85,B 0,C 180,E1 12067.179,E2 12067.179} C_VEL
LIN {X 0,Y 362.029,Z 685.03,A -85,B 0,C 180,E1 12074.487,E2 12074.487} C_VEL
LIN {X 0,Y 361.674,Z 685.03,A -85,B 0,C 180,E1 12082.059,E2 12082.059} C_VEL
LIN {X 0,Y 361.33,Z 685.03,A -85,B 0,C 180,E1 12090.079,E2 12090.079} C_VEL
LIN {X 0,Y 361.369,Z 685.672,A -85,B 0,C 180,E1 12097.995,E2 12097.995} C_VEL
LIN {X 0,Y 370.1,Z 708.678,A -85,B 0,C 180,E1 12101.109,E2 12101.109} C_VEL
LIN {X 0,Y 393.072,Z 757.933,A -85,B 0,C 180,E1 12105.273,E2 12105.273} C_VEL
LIN {X 0,Y 399.437,Z 776.178,A -85,B 0,C 180,E1 12106.695,E2 12106.695} C_VEL
LIN {X 0,Y 393.634,Z 818.877,A -85,B 0,C 180,E1 12108.81,E2 12108.81} C_VEL
LIN {X 0,Y 386.903,Z 858.08,A -85,B 0,C 180,E1 12111.747,E2 12111.747} C_VEL
LIN {X 0,Y 380.369,Z 892.939,A -85,B 0,C 180,E1 12115.405,E2 12115.405} C_VEL
LIN {X 0,Y 374.242,Z 924.228,A -85,B 0,C 180,E1 12119.849,E2 12119.849} C_VEL
LIN {X 0,Y 369.151,Z 951.283,A -85,B 0,C 180,E1 12125.043,E2 12125.043} C_VEL
LIN {X 0,Y 365.711,Z 972.824,A -85,B 0,C 180,E1 12130.728,E2 12130.728} C_VEL
LIN {X 0,Y 364.031,Z 988.324,A -85,B 0,C 180,E1 12136.598,E2 12136.598} C_VEL
LIN {X 0,Y 363.538,Z 996.915,A -85,B 0,C 180,E1 12141.65,E2 12141.65} C_VEL
LIN {X 0,Y 363.466,Z 1000.52,A -85,B 0,C 180,E1 12145.24,E2 12145.24} C_VEL
LIN {X 0,Y 363.526,Z 1002.118,A -85,B 0,C 180,E1 12150.004,E2 12150.004} C_VEL
LIN {X 0,Y 363.558,Z 999.008,A -85,B 0,C 180,E1 12155.84,E2 12155.84} C_VEL
LIN {X 0,Y 363.703,Z 994.533,A -85,B 0,C 180,E1 12159.286,E2 12159.286} C_VEL
LIN {X 0,Y 361.398,Z 990.917,A -85,B 0,C 180,E1 12161.247,E2 12161.247} C_VEL
LIN {X 0,Y 356.495,Z 984.221,A -85,B 0,C 180,E1 12164.14,E2 12164.14} C_VEL
LIN {X 0,Y 356.46,Z 983.41,A -85,B 0,C 180,E1 12164.471,E2 12164.471} C_VEL
LIN {X 0,Y 358.233,Z 967.22,A -85,B 0,C 180,E1 12170.019,E2 12170.019} C_VEL
LIN {X 0,Y 361.628,Z 944.005,A -85,B 0,C 180,E1 12175.684,E2 12175.684} C_VEL
LIN {X 0,Y 366.75,Z 914.412,A -85,B 0,C 180,E1 12180.982,E2 12180.982} C_VEL
LIN {X 0,Y 373.24,Z 879.431,A -85,B 0,C 180,E1 12185.654,E2 12185.654} C_VEL
LIN {X 0,Y 381.016,Z 838.549,A -85,B 0,C 180,E1 12189.696,E2 12189.696} C_VEL
LIN {X 0,Y 389.268,Z 794.049,A -85,B 0,C 180,E1 12192.831,E2 12192.831} C_VEL
LIN {X 0,Y 392.317,Z 774.831,A -85,B 0,C 180,E1 12193.915,E2 12193.915} C_VEL
LIN {X 0,Y 388.003,Z 742.825,A -85,B 0,C 180,E1 12197.378,E2 12197.378} C_VEL
LIN {X 0,Y 384.98,Z 731.236,A -85,B 0,C 180,E1 12199.588,E2 12199.588} C_VEL
LIN {X 0,Y 383.276,Z 727.731,A -85,B 0,C 180,E1 12200.952,E2 12200.952} C_VEL
LIN {X 0,Y 381.301,Z 725.352,A -85,B 0,C 180,E1 12203.583,E2 12203.583} C_VEL
LIN {X 0,Y 381.895,Z 727.938,A -85,B 0,C 180,E1 12206.995,E2 12206.995} C_VEL
LIN {X 0,Y 384.541,Z 737.195,A -85,B 0,C 180,E1 12210.026,E2 12210.026} C_VEL
LIN {X 0,Y 386.61,Z 745.778,A -85,B 0,C 180,E1 12211.68,E2 12211.68} C_VEL
LIN {X 0,Y 377.838,Z 797.608,A -85,B 0,C 180,E1 12214.888,E2 12214.888} C_VEL
LIN {X 0,Y 373.409,Z 825.956,A -85,B 0,C 180,E1 12217.577,E2 12217.577} C_VEL
LIN {X 0,Y 368.889,Z 849.13,A -85,B 0,C 180,E1 12220.894,E2 12220.894} C_VEL
LIN {X 0,Y 364.782,Z 867.028,A -85,B 0,C 180,E1 12224.705,E2 12224.705} C_VEL
LIN {X 0,Y 361.37,Z 880.231,A -85,B 0,C 180,E1 12229.076,E2 12229.076} C_VEL
LIN {X 0,Y 359.13,Z 888.068,A -85,B 0,C 180,E1 12233.965,E2 12233.965} C_VEL
LIN {X 0,Y 358.246,Z 889.961,A -85,B 0,C 180,E1 12237.581,E2 12237.581} C_VEL
LIN {X 0,Y 357.882,Z 887.475,A -85,B 0,C 180,E1 12242.411,E2 12242.411} C_VEL
LIN {X 0,Y 358.118,Z 880.523,A -85,B 0,C 180,E1 12246.648,E2 12246.648} C_VEL
LIN {X 0,Y 359.322,Z 867.38,A -85,B 0,C 180,E1 12251.193,E2 12251.193} C_VEL
LIN {X 0,Y 361.388,Z 848.836,A -85,B 0,C 180,E1 12255.312,E2 12255.312} C_VEL
LIN {X 0,Y 363.954,Z 826.182,A -85,B 0,C 180,E1 12258.736,E2 12258.736} C_VEL
LIN {X 0,Y 366.567,Z 798.255,A -85,B 0,C 180,E1 12261.58,E2 12261.58} C_VEL
LIN {X 0,Y 368.606,Z 769.051,A -85,B 0,C 180,E1 12263.435,E2 12263.435} C_VEL
LIN {X 0,Y 369.371,Z 731.399,A -85,B 0,C 180,E1 12264.767,E2 12264.767} C_VEL
LIN {X 0,Y 353.515,Z 685.03,A -85,B 0,C 180,E1 12267.561,E2 12267.561} C_VEL
LIN {X 0,Y 353.331,Z 685.03,A -85,B 0,C 180,E1 12275.752,E2 12275.752} C_VEL
LIN {X 0,Y 353.235,Z 685.03,A -85,B 0,C 180,E1 12283.107,E2 12283.107} C_VEL
LIN {X 0,Y 353.279,Z 685.03,A -85,B 0,C 180,E1 12290.237,E2 12290.237} C_VEL
LIN {X 0,Y 353.399,Z 685.03,A -85,B 0,C 180,E1 12292.728,E2 12292.728} C_VEL
LIN {X 0,Y 357.866,Z 694.933,A -85,B 0,C 180,E1 12293.542,E2 12293.542} C_VEL
LIN {X 0,Y 372.91,Z 727.553,A -85,B 0,C 180,E1 12296.296,E2 12296.296} C_VEL
LIN {X 0,Y 380.104,Z 751.742,A -85,B 0,C 180,E1 12298.447,E2 12298.447} C_VEL
LIN {X 0,Y 376.401,Z 782.842,A -85,B 0,C 180,E1 12300.787,E2 12300.787} C_VEL
LIN {X 0,Y 371.788,Z 811.187,A -85,B 0,C 180,E1 12303.964,E2 12303.964} C_VEL
LIN {X 0,Y 366.94,Z 835.371,A -85,B 0,C 180,E1 12307.833,E2 12307.833} C_VEL
LIN {X 0,Y 362.624,Z 855.388,A -85,B 0,C 180,E1 12312.436,E2 12312.436} C_VEL
LIN {X 0,Y 359.679,Z 869.506,A -85,B 0,C 180,E1 12317.271,E2 12317.271} C_VEL
LIN {X 0,Y 357.862,Z 879.282,A -85,B 0,C 180,E1 12322.728,E2 12322.728} C_VEL
LIN {X 0,Y 357.219,Z 883.276,A -85,B 0,C 180,E1 12327.575,E2 12327.575} C_VEL
LIN {X 0,Y 357.218,Z 883.24,A -85,B 0,C 180,E1 12332.418,E2 12332.418} C_VEL
LIN {X 0,Y 357.882,Z 879.172,A -85,B 0,C 180,E1 12337.264,E2 12337.264} C_VEL
LIN {X 0,Y 359.694,Z 869.295,A -85,B 0,C 180,E1 12342.721,E2 12342.721} C_VEL
LIN {X 0,Y 362.911,Z 853.923,A -85,B 0,C 180,E1 12347.855,E2 12347.855} C_VEL
LIN {X 0,Y 367.072,Z 834.706,A -85,B 0,C 180,E1 12352.196,E2 12352.196} C_VEL
LIN {X 0,Y 371.878,Z 810.547,A -85,B 0,C 180,E1 12356.022,E2 12356.022} C_VEL
LIN {X 0,Y 376.414,Z 782.016,A -85,B 0,C 180,E1 12359.194,E2 12359.194} C_VEL
LIN {X 0,Y 379.963,Z 751.067,A -85,B 0,C 180,E1 12361.513,E2 12361.513} C_VEL
LIN {X 0,Y 370.606,Z 721.905,A -85,B 0,C 180,E1 12364.088,E2 12364.088} C_VEL
LIN {X 0,Y 354.836,Z 689.575,A -85,B 0,C 180,E1 12366.858,E2 12366.858} C_VEL
LIN {X 0,Y 353.379,Z 685.03,A -85,B 0,C 180,E1 12367.2,E2 12367.2} C_VEL
LIN {X 0,Y 353.188,Z 685.03,A -85,B 0,C 180,E1 12373.434,E2 12373.434} C_VEL
LIN {X 0,Y 353.265,Z 685.03,A -85,B 0,C 180,E1 12380.252,E2 12380.252} C_VEL
LIN {X 0,Y 353.31,Z 685.03,A -85,B 0,C 180,E1 12386.283,E2 12386.283} C_VEL
LIN {X 0,Y 353.513,Z 685.03,A -85,B 0,C 180,E1 12393.687,E2 12393.687} C_VEL
LIN {X 0,Y 353.883,Z 685.03,A -85,B 0,C 180,E1 12400.062,E2 12400.062} C_VEL
LIN {X 0,Y 354.368,Z 685.03,A -85,B 0,C 180,E1 12407.713,E2 12407.713} C_VEL
LIN {X 0,Y 354.697,Z 685.03,A -85,B 0,C 180,E1 12415.125,E2 12415.125} C_VEL
LIN {X 0,Y 354.935,Z 685.03,A -85,B 0,C 180,E1 12422.442,E2 12422.442} C_VEL
LIN {X 0,Y 354.323,Z 685.03,A -85,B 0,C 180,E1 12429.813,E2 12429.813} C_VEL
LIN {X 0,Y 353.972,Z 685.03,A -85,B 0,C 180,E1 12437.366,E2 12437.366} C_VEL
LIN {X 0,Y 353.565,Z 685.03,A -85,B 0,C 180,E1 12445.268,E2 12445.268} C_VEL
LIN {X 0,Y 353.311,Z 685.03,A -85,B 0,C 180,E1 12451.33,E2 12451.33} C_VEL
LIN {X 0,Y 353.343,Z 685.064,A -85,B 0,C 180,E1 12456.939,E2 12456.939} C_VEL
LIN {X 0,Y 361.954,Z 707.849,A -85,B 0,C 180,E1 12460.101,E2 12460.101} C_VEL
LIN {X 0,Y 385.184,Z 757.57,A -85,B 0,C 180,E1 12464.451,E2 12464.451} C_VEL
LIN {X 0,Y 392.692,Z 777.606,A -85,B 0,C 180,E1 12466.124,E2 12466.124} C_VEL
LIN {X 0,Y 386.876,Z 818.274,A -85,B 0,C 180,E1 12468.189,E2 12468.189} C_VEL
LIN {X 0,Y 380.056,Z 856.767,A -85,B 0,C 180,E1 12471.112,E2 12471.112} C_VEL
LIN {X 0,Y 373.042,Z 892.699,A -85,B 0,C 180,E1 12474.937,E2 12474.937} C_VEL
LIN {X 0,Y 366.639,Z 924.231,A -85,B 0,C 180,E1 12479.522,E2 12479.522} C_VEL
LIN {X 0,Y 361.403,Z 950.965,A -85,B 0,C 180,E1 12484.79,E2 12484.79} C_VEL
LIN {X 0,Y 358.014,Z 971.443,A -85,B 0,C 180,E1 12490.297,E2 12490.297} C_VEL
LIN {X 0,Y 356.194,Z 987.118,A -85,B 0,C 180,E1 12496.308,E2 12496.308} C_VEL
LIN {X 0,Y 355.693,Z 995.769,A -85,B 0,C 180,E1 12501.464,E2 12501.464} C_VEL
LIN {X 0,Y 355.625,Z 999.403,A -85,B 0,C 180,E1 12505.135,E2 12505.135} C_VEL
LIN {X 0,Y 355.711,Z 1000.995,A -85,B 0,C 180,E1 12510.004,E2 12510.004} C_VEL
LIN {X 0,Y 355.693,Z 998.828,A -85,B 0,C 180,E1 12514.871,E2 12514.871} C_VEL
LIN {X 0,Y 355.924,Z 991.845,A -85,B 0,C 180,E1 12520.385,E2 12520.385} C_VEL
LIN {X 0,Y 356.46,Z 983.41,A -85,B 0,C 180,E1 12524.471,E2 12524.471} C_VEL
LIN {X 0,Y 355.474,Z 980.076,A -85,B 0,C 180,E1 12525.767,E2 12525.767} C_VEL
LIN {X 0,Y 350.064,Z 969.8,A -85,B 0,C 180,E1 12529.238,E2 12529.238} C_VEL
LIN {X 0,Y 350.119,Z 968.753,A -85,B 0,C 180,E1 12529.557,E2 12529.557} C_VEL
LIN {X 0,Y 353.347,Z 946.85,A -85,B 0,C 180,E1 12535.287,E2 12535.287} C_VEL
LIN {X 0,Y 358.283,Z 919.48,A -85,B 0,C 180,E1 12540.571,E2 12540.571} C_VEL
LIN {X 0,Y 365.095,Z 884.771,A -85,B 0,C 180,E1 12545.576,E2 12545.576} C_VEL
LIN {X 0,Y 373.332,Z 844.668,A -85,B 0,C 180,E1 12549.859,E2 12549.859} C_VEL
LIN {X 0,Y 382.441,Z 799.888,A -85,B 0,C 180,E1 12553.299,E2 12553.299} C_VEL
LIN {X 0,Y 386.517,Z 777.511,A -85,B 0,C 180,E1 12554.655,E2 12554.655} C_VEL
LIN {X 0,Y 383.578,Z 746.522,A -85,B 0,C 180,E1 12558.23,E2 12558.23} C_VEL
LIN {X 0,Y 381.453,Z 737.36,A -85,B 0,C 180,E1 12560.189,E2 12560.189} C_VEL
LIN {X 0,Y 378.927,Z 733.298,A -85,B 0,C 180,E1 12562.803,E2 12562.803} C_VEL
LIN {X 0,Y 378.78,Z 735.129,A -85,B 0,C 180,E1 12566.795,E2 12566.795} C_VEL
LIN {X 0,Y 380.556,Z 743.148,A -85,B 0,C 180,E1 12569.527,E2 12569.527} C_VEL
LIN {X 0,Y 381.601,Z 750.407,A -85,B 0,C 180,E1 12570.924,E2 12570.924} C_VEL
LIN {X 0,Y 372.233,Z 797.739,A -85,B 0,C 180,E1 12573.999,E2 12573.999} C_VEL
LIN {X 0,Y 367.35,Z 826.159,A -85,B 0,C 180,E1 12576.707,E2 12576.707} C_VEL
LIN {X 0,Y 362.306,Z 850.106,A -85,B 0,C 180,E1 12580.18,E2 12580.18} C_VEL
LIN {X 0,Y 357.803,Z 868.22,A -85,B 0,C 180,E1 12584.086,E2 12584.086} C_VEL
LIN {X 0,Y 353.91,Z 881.953,A -85,B 0,C 180,E1 12588.751,E2 12588.751} C_VEL
LIN {X 0,Y 351.449,Z 889.728,A -85,B 0,C 180,E1 12593.833,E2 12593.833} C_VEL
LIN {X 0,Y 350.494,Z 891.437,A -85,B 0,C 180,E1 12597.527,E2 12597.527} C_VEL
LIN {X 0,Y 350.115,Z 888.752,A -85,B 0,C 180,E1 12602.464,E2 12602.464} C_VEL
LIN {X 0,Y 350.349,Z 881.609,A -85,B 0,C 180,E1 12606.796,E2 12606.796} C_VEL
LIN {X 0,Y 351.607,Z 868.213,A -85,B 0,C 180,E1 12611.442,E2 12611.442} C_VEL
LIN {X 0,Y 353.84,Z 849.018,A -85,B 0,C 180,E1 12615.735,E2 12615.735} C_VEL
LIN {X 0,Y 356.621,Z 825.32,A -85,B 0,C 180,E1 12619.296,E2 12619.296} C_VEL
LIN {X 0,Y 359.208,Z 798.265,A -85,B 0,C 180,E1 12622.045,E2 12622.045} C_VEL
LIN {X 0,Y 361.339,Z 768.354,A -85,B 0,C 180,E1 12623.938,E2 12623.938} C_VEL
LIN {X 0,Y 362.11,Z 733.179,A -85,B 0,C 180,E1 12625.202,E2 12625.202} C_VEL
LIN {X 0,Y 345.503,Z 685.03,A -85,B 0,C 180,E1 12628.318,E2 12628.318} C_VEL
LIN {X 0,Y 345.361,Z 685.03,A -85,B 0,C 180,E1 12634.602,E2 12634.602} C_VEL
LIN {X 0,Y 345.241,Z 685.03,A -85,B 0,C 180,E1 12641.999,E2 12641.999} C_VEL
LIN {X 0,Y 345.232,Z 685.03,A -85,B 0,C 180,E1 12649.024,E2 12649.024} C_VEL
LIN {X 0,Y 345.458,Z 685.03,A -85,B 0,C 180,E1 12651.651,E2 12651.651} C_VEL
LIN {X 0,Y 351.665,Z 698.207,A -85,B 0,C 180,E1 12652.848,E2 12652.848} C_VEL
LIN {X 0,Y 365.867,Z 728.916,A -85,B 0,C 180,E1 12655.561,E2 12655.561} C_VEL
LIN {X 0,Y 373.284,Z 754.585,A -85,B 0,C 180,E1 12657.923,E2 12657.923} C_VEL
LIN {X 0,Y 369.438,Z 785.282,A -85,B 0,C 180,E1 12660.308,E2 12660.308} C_VEL
LIN {X 0,Y 364.537,Z 813.521,A -85,B 0,C 180,E1 12663.571,E2 12663.571} C_VEL
LIN {X 0,Y 359.607,Z 837.077,A -85,B 0,C 180,E1 12667.456,E2 12667.456} C_VEL
LIN {X 0,Y 355.172,Z 856.633,A -85,B 0,C 180,E1 12672.055,E2 12672.055} C_VEL
LIN {X 0,Y 352.049,Z 870.755,A -85,B 0,C 180,E1 12676.991,E2 12676.991} C_VEL
LIN {X 0,Y 350.122,Z 880.529,A -85,B 0,C 180,E1 12682.567,E2 12682.567} C_VEL
LIN {X 0,Y 349.431,Z 884.522,A -85,B 0,C 180,E1 12687.521,E2 12687.521} C_VEL
LIN {X 0,Y 349.431,Z 884.486,A -85,B 0,C 180,E1 12692.471,E2 12692.471} C_VEL
LIN {X 0,Y 350.236,Z 879.974,A -85,B 0,C 180,E1 12697.787,E2 12697.787} C_VEL
LIN {X 0,Y 352.064,Z 870.547,A -85,B 0,C 180,E1 12703.001,E2 12703.001} C_VEL
LIN {X 0,Y 355.494,Z 855.169,A -85,B 0,C 180,E1 12708.24,E2 12708.24} C_VEL
LIN {X 0,Y 359.965,Z 835.441,A -85,B 0,C 180,E1 12712.767,E2 12712.767} C_VEL
LIN {X 0,Y 365.056,Z 810.703,A -85,B 0,C 180,E1 12716.711,E2 12716.711} C_VEL
LIN {X 0,Y 369.721,Z 782.743,A -85,B 0,C 180,E1 12719.828,E2 12719.828} C_VEL
LIN {X 0,Y 373.04,Z 752.511,A -85,B 0,C 180,E1 12722.155,E2 12722.155} C_VEL
LIN {X 0,Y 363.429,Z 722.66,A -85,B 0,C 180,E1 12724.88,E2 12724.88} C_VEL
LIN {X 0,Y 346.901,Z 689.656,A -85,B 0,C 180,E1 12727.883,E2 12727.883} C_VEL
LIN {X 0,Y 345.342,Z 685.03,A -85,B 0,C 180,E1 12728.241,E2 12728.241} C_VEL
LIN {X 0,Y 345.201,Z 685.03,A -85,B 0,C 180,E1 12735.632,E2 12735.632} C_VEL
LIN {X 0,Y 345.259,Z 685.03,A -85,B 0,C 180,E1 12742.285,E2 12742.285} C_VEL
LIN {X 0,Y 345.43,Z 685.03,A -85,B 0,C 180,E1 12748.394,E2 12748.394} C_VEL
LIN {X 0,Y 345.729,Z 685.03,A -85,B 0,C 180,E1 12756.429,E2 12756.429} C_VEL
LIN {X 0,Y 346.158,Z 685.03,A -85,B 0,C 180,E1 12763.542,E2 12763.542} C_VEL
LIN {X 0,Y 346.482,Z 685.03,A -85,B 0,C 180,E1 12769.974,E2 12769.974} C_VEL
LIN {X 0,Y 346.939,Z 685.03,A -85,B 0,C 180,E1 12777.513,E2 12777.513} C_VEL
LIN {X 0,Y 347.037,Z 685.03,A -85,B 0,C 180,E1 12782.497,E2 12782.497} C_VEL
LIN {X 0,Y 346.399,Z 685.03,A -85,B 0,C 180,E1 12790.04,E2 12790.04} C_VEL
LIN {X 0,Y 346,Z 685.03,A -85,B 0,C 180,E1 12797.78,E2 12797.78} C_VEL
LIN {X 0,Y 345.621,Z 685.03,A -85,B 0,C 180,E1 12805.891,E2 12805.891} C_VEL
LIN {X 0,Y 345.389,Z 685.03,A -85,B 0,C 180,E1 12813.892,E2 12813.892} C_VEL
LIN {X 0,Y 345.465,Z 685.425,A -85,B 0,C 180,E1 12815.967,E2 12815.967} C_VEL
LIN {X 0,Y 353.751,Z 706.985,A -85,B 0,C 180,E1 12819.042,E2 12819.042} C_VEL
LIN {X 0,Y 377.633,Z 757.912,A -85,B 0,C 180,E1 12823.67,E2 12823.67} C_VEL
LIN {X 0,Y 385.663,Z 780.945,A -85,B 0,C 180,E1 12825.629,E2 12825.629} C_VEL
LIN {X 0,Y 379.579,Z 820.902,A -85,B 0,C 180,E1 12827.773,E2 12827.773} C_VEL
LIN {X 0,Y 372.396,Z 859.455,A -85,B 0,C 180,E1 12830.834,E2 12830.834} C_VEL
LIN {X 0,Y 365.372,Z 894.148,A -85,B 0,C 180,E1 12834.678,E2 12834.678} C_VEL
LIN {X 0,Y 358.675,Z 925.768,A -85,B 0,C 180,E1 12839.469,E2 12839.469} C_VEL
LIN {X 0,Y 353.499,Z 951.44,A -85,B 0,C 180,E1 12844.733,E2 12844.733} C_VEL
LIN {X 0,Y 350.066,Z 971.617,A -85,B 0,C 180,E1 12850.377,E2 12850.377} C_VEL
LIN {X 0,Y 348.409,Z 985.608,A -85,B 0,C 180,E1 12855.875,E2 12855.875} C_VEL
LIN {X 0,Y 347.868,Z 994.603,A -85,B 0,C 180,E1 12861.271,E2 12861.271} C_VEL
LIN {X 0,Y 347.728,Z 999.099,A -85,B 0,C 180,E1 12866.484,E2 12866.484} C_VEL
LIN {X 0,Y 347.891,Z 999.857,A -85,B 0,C 180,E1 12870.004,E2 12870.004} C_VEL
LIN {X 0,Y 347.881,Z 997.651,A -85,B 0,C 180,E1 12874.981,E2 12874.981} C_VEL
LIN {X 0,Y 348.121,Z 990.582,A -85,B 0,C 180,E1 12880.62,E2 12880.62} C_VEL
LIN {X 0,Y 349.048,Z 978.235,A -85,B 0,C 180,E1 12886.325,E2 12886.325} C_VEL
LIN {X 0,Y 350.119,Z 968.753,A -85,B 0,C 180,E1 12889.557,E2 12889.557} C_VEL
LIN {X 0,Y 349.475,Z 964.573,A -85,B 0,C 180,E1 12890.812,E2 12890.812} C_VEL
LIN {X 0,Y 344.808,Z 952.334,A -85,B 0,C 180,E1 12894.19,E2 12894.19} C_VEL
LIN {X 0,Y 344.923,Z 951.12,A -85,B 0,C 180,E1 12894.495,E2 12894.495} C_VEL
LIN {X 0,Y 350.084,Z 923.124,A -85,B 0,C 180,E1 12900.346,E2 12900.346} C_VEL
LIN {X 0,Y 356.984,Z 889.566,A -85,B 0,C 180,E1 12905.543,E2 12905.543} C_VEL
LIN {X 0,Y 365.674,Z 850.206,A -85,B 0,C 180,E1 12910.068,E2 12910.068} C_VEL
LIN {X 0,Y 375.715,Z 805.413,A -85,B 0,C 180,E1 12913.793,E2 12913.793} C_VEL
LIN {X 0,Y 381.079,Z 781.378,A -85,B 0,C 180,E1 12915.281,E2 12915.281} C_VEL
LIN {X 0,Y 379.459,Z 751.309,A -85,B 0,C 180,E1 12918.944,E2 12918.944} C_VEL
LIN {X 0,Y 377.954,Z 743.361,A -85,B 0,C 180,E1 12920.808,E2 12920.808} C_VEL
LIN {X 0,Y 375.765,Z 740.409,A -85,B 0,C 180,E1 12923.443,E2 12923.443} C_VEL
LIN {X 0,Y 375.589,Z 742.077,A -85,B 0,C 180,E1 12926.475,E2 12926.475} C_VEL
LIN {X 0,Y 376.806,Z 750.215,A -85,B 0,C 180,E1 12929.296,E2 12929.296} C_VEL
LIN {X 0,Y 377.231,Z 753.468,A -85,B 0,C 180,E1 12930.008,E2 12930.008} C_VEL
LIN {X 0,Y 366.557,Z 800.308,A -85,B 0,C 180,E1 12933.236,E2 12933.236} C_VEL
LIN {X 0,Y 360.975,Z 828.972,A -85,B 0,C 180,E1 12936.107,E2 12936.107} C_VEL
LIN {X 0,Y 355.533,Z 852.318,A -85,B 0,C 180,E1 12939.641,E2 12939.641} C_VEL
LIN {X 0,Y 350.552,Z 870.595,A -85,B 0,C 180,E1 12943.747,E2 12943.747} C_VEL
LIN {X 0,Y 346.443,Z 883.928,A -85,B 0,C 180,E1 12948.505,E2 12948.505} C_VEL
LIN {X 0,Y 343.778,Z 891.411,A -85,B 0,C 180,E1 12953.695,E2 12953.695} C_VEL
LIN {X 0,Y 342.763,Z 892.909,A -85,B 0,C 180,E1 12957.471,E2 12957.471} C_VEL
LIN {X 0,Y 342.321,Z 890.018,A -85,B 0,C 180,E1 12962.521,E2 12962.521} C_VEL
LIN {X 0,Y 342.704,Z 881.216,A -85,B 0,C 180,E1 12967.584,E2 12967.584} C_VEL
LIN {X 0,Y 344.172,Z 866.737,A -85,B 0,C 180,E1 12972.335,E2 12972.335} C_VEL
LIN {X 0,Y 346.539,Z 847.06,A -85,B 0,C 180,E1 12976.536,E2 12976.536} C_VEL
LIN {X 0,Y 349.441,Z 823.016,A -85,B 0,C 180,E1 12980.038,E2 12980.038} C_VEL
LIN {X 0,Y 352.193,Z 794.72,A -85,B 0,C 180,E1 12982.796,E2 12982.796} C_VEL
LIN {X 0,Y 354.227,Z 764.672,A -85,B 0,C 180,E1 12984.593,E2 12984.593} C_VEL
LIN {X 0,Y 354.673,Z 734.208,A -85,B 0,C 180,E1 12985.695,E2 12985.695} C_VEL
LIN {X 0,Y 337.538,Z 685.03,A -85,B 0,C 180,E1 12988.969,E2 12988.969} C_VEL
LIN {X 0,Y 337.301,Z 685.03,A -85,B 0,C 180,E1 12996.352,E2 12996.352} C_VEL
LIN {X 0,Y 337.351,Z 685.03,A -85,B 0,C 180,E1 13002.129,E2 13002.129} C_VEL
LIN {X 0,Y 337.381,Z 685.03,A -85,B 0,C 180,E1 13009.481,E2 13009.481} C_VEL
LIN {X 0,Y 337.497,Z 685.03,A -85,B 0,C 180,E1 13010.559,E2 13010.559} C_VEL
LIN {X 0,Y 341.747,Z 694.555,A -85,B 0,C 180,E1 13011.434,E2 13011.434} C_VEL
LIN {X 0,Y 357.792,Z 727.211,A -85,B 0,C 180,E1 13014.523,E2 13014.523} C_VEL
LIN {X 0,Y 366.468,Z 755.302,A -85,B 0,C 180,E1 13017.211,E2 13017.211} C_VEL
LIN {X 0,Y 362.601,Z 786.977,A -85,B 0,C 180,E1 13019.74,E2 13019.74} C_VEL
LIN {X 0,Y 357.573,Z 814.753,A -85,B 0,C 180,E1 13023.015,E2 13023.015} C_VEL
LIN {X 0,Y 352.318,Z 838.744,A -85,B 0,C 180,E1 13027.058,E2 13027.058} C_VEL
LIN {X 0,Y 347.505,Z 858.91,A -85,B 0,C 180,E1 13031.972,E2 13031.972} C_VEL
LIN {X 0,Y 344.129,Z 873.427,A -85,B 0,C 180,E1 13037.33,E2 13037.33} C_VEL
LIN {X 0,Y 342.396,Z 881.774,A -85,B 0,C 180,E1 13042.398,E2 13042.398} C_VEL
LIN {X 0,Y 341.632,Z 885.77,A -85,B 0,C 180,E1 13047.464,E2 13047.464} C_VEL
LIN {X 0,Y 341.633,Z 885.735,A -85,B 0,C 180,E1 13052.528,E2 13052.528} C_VEL
LIN {X 0,Y 342.421,Z 881.666,A -85,B 0,C 180,E1 13057.594,E2 13057.594} C_VEL
LIN {X 0,Y 344.446,Z 871.797,A -85,B 0,C 180,E1 13063.294,E2 13063.294} C_VEL
LIN {X 0,Y 348.105,Z 856.414,A -85,B 0,C 180,E1 13068.642,E2 13068.642} C_VEL
LIN {X 0,Y 352.776,Z 836.687,A -85,B 0,C 180,E1 13073.258,E2 13073.258} C_VEL
LIN {X 0,Y 358.111,Z 811.942,A -85,B 0,C 180,E1 13077.272,E2 13077.272} C_VEL
LIN {X 0,Y 363.081,Z 783.445,A -85,B 0,C 180,E1 13080.486,E2 13080.486} C_VEL
LIN {X 0,Y 366.388,Z 755.072,A -85,B 0,C 180,E1 13082.709,E2 13082.709} C_VEL
LIN {X 0,Y 357.252,Z 725.951,A -85,B 0,C 180,E1 13085.486,E2 13085.486} C_VEL
LIN {X 0,Y 341.242,Z 693.789,A -85,B 0,C 180,E1 13088.543,E2 13088.543} C_VEL
LIN {X 0,Y 337.425,Z 685.03,A -85,B 0,C 180,E1 13089.429,E2 13089.429} C_VEL
LIN {X 0,Y 337.292,Z 685.03,A -85,B 0,C 180,E1 13095.708,E2 13095.708} C_VEL
LIN {X 0,Y 337.321,Z 685.03,A -85,B 0,C 180,E1 13103.63,E2 13103.63} C_VEL
LIN {X 0,Y 337.528,Z 685.03,A -85,B 0,C 180,E1 13110.552,E2 13110.552} C_VEL
LIN {X 0,Y 337.823,Z 685.03,A -85,B 0,C 180,E1 13116.304,E2 13116.304} C_VEL
LIN {X 0,Y 338.112,Z 685.03,A -85,B 0,C 180,E1 13121.803,E2 13121.803} C_VEL
LIN {X 0,Y 338.546,Z 685.03,A -85,B 0,C 180,E1 13129.736,E2 13129.736} C_VEL
LIN {X 0,Y 339.026,Z 685.03,A -85,B 0,C 180,E1 13137.455,E2 13137.455} C_VEL
LIN {X 0,Y 339.118,Z 685.03,A -85,B 0,C 180,E1 13142.556,E2 13142.556} C_VEL
LIN {X 0,Y 338.459,Z 685.03,A -85,B 0,C 180,E1 13150.278,E2 13150.278} C_VEL
LIN {X 0,Y 338.028,Z 685.03,A -85,B 0,C 180,E1 13158.214,E2 13158.214} C_VEL
LIN {X 0,Y 337.796,Z 685.03,A -85,B 0,C 180,E1 13163.71,E2 13163.71} C_VEL
LIN {X 0,Y 337.488,Z 685.03,A -85,B 0,C 180,E1 13171.841,E2 13171.841} C_VEL
LIN {X 0,Y 337.489,Z 685.48,A -85,B 0,C 180,E1 13174.915,E2 13174.915} C_VEL
LIN {X 0,Y 345.45,Z 705.977,A -85,B 0,C 180,E1 13177.936,E2 13177.936} C_VEL
LIN {X 0,Y 369.711,Z 757.448,A -85,B 0,C 180,E1 13182.8,E2 13182.8} C_VEL
LIN {X 0,Y 378.793,Z 782.622,A -85,B 0,C 180,E1 13185.056,E2 13185.056} C_VEL
LIN {X 0,Y 372.287,Z 823.398,A -85,B 0,C 180,E1 13187.341,E2 13187.341} C_VEL
LIN {X 0,Y 364.63,Z 862.892,A -85,B 0,C 180,E1 13190.628,E2 13190.628} C_VEL
LIN {X 0,Y 356.905,Z 898.965,A -85,B 0,C 180,E1 13194.889,E2 13194.889} C_VEL
LIN {X 0,Y 350.143,Z 929.892,A -85,B 0,C 180,E1 13199.914,E2 13199.914} C_VEL
LIN {X 0,Y 345.022,Z 954.924,A -85,B 0,C 180,E1 13205.452,E2 13205.452} C_VEL
LIN {X 0,Y 341.701,Z 974.273,A -85,B 0,C 180,E1 13211.366,E2 13211.366} C_VEL
LIN {X 0,Y 340.324,Z 987.658,A -85,B 0,C 180,E1 13217.29,E2 13217.29} C_VEL
LIN {X 0,Y 340.031,Z 994.893,A -85,B 0,C 180,E1 13222.353,E2 13222.353} C_VEL
LIN {X 0,Y 339.969,Z 998.385,A -85,B 0,C 180,E1 13227.46,E2 13227.46} C_VEL
LIN {X 0,Y 340.038,Z 998.061,A -85,B 0,C 180,E1 13232.547,E2 13232.547} C_VEL
LIN {X 0,Y 340.136,Z 993.913,A -85,B 0,C 180,E1 13237.653,E2 13237.653} C_VEL
LIN {X 0,Y 340.615,Z 984.62,A -85,B 0,C 180,E1 13243.388,E2 13243.388} C_VEL
LIN {X 0,Y 342.278,Z 968.356,A -85,B 0,C 180,E1 13249.689,E2 13249.689} C_VEL
LIN {X 0,Y 344.923,Z 951.12,A -85,B 0,C 180,E1 13254.495,E2 13254.495} C_VEL
LIN {X 0,Y 342.895,Z 941.412,A -85,B 0,C 180,E1 13256.901,E2 13256.901} C_VEL
LIN {X 0,Y 340.989,Z 930.971,A -85,B 0,C 180,E1 13259.252,E2 13259.252} C_VEL
LIN {X 0,Y 347.78,Z 899.504,A -85,B 0,C 180,E1 13264.721,E2 13264.721} C_VEL
LIN {X 0,Y 356.722,Z 861.5,A -85,B 0,C 180,E1 13269.634,E2 13269.634} C_VEL
LIN {X 0,Y 366.774,Z 820.204,A -85,B 0,C 180,E1 13273.57,E2 13273.57} C_VEL
LIN {X 0,Y 375.515,Z 782.858,A -85,B 0,C 180,E1 13276.242,E2 13276.242} C_VEL
LIN {X 0,Y 375.49,Z 757.224,A -85,B 0,C 180,E1 13279.491,E2 13279.491} C_VEL
LIN {X 0,Y 374.766,Z 750.715,A -85,B 0,C 180,E1 13280.966,E2 13280.966} C_VEL
LIN {X 0,Y 373.259,Z 748.243,A -85,B 0,C 180,E1 13282.666,E2 13282.666} C_VEL
LIN {X 0,Y 372.248,Z 748.38,A -85,B 0,C 180,E1 13285.419,E2 13285.419} C_VEL
LIN {X 0,Y 372.608,Z 752.611,A -85,B 0,C 180,E1 13287.723,E2 13287.723} C_VEL
LIN {X 0,Y 372.701,Z 758.419,A -85,B 0,C 180,E1 13289.156,E2 13289.156} C_VEL
LIN {X 0,Y 361.059,Z 803.292,A -85,B 0,C 180,E1 13292.458,E2 13292.458} C_VEL
LIN {X 0,Y 354.7,Z 831.947,A -85,B 0,C 180,E1 13295.49,E2 13295.49} C_VEL
LIN {X 0,Y 348.641,Z 855.377,A -85,B 0,C 180,E1 13299.22,E2 13299.22} C_VEL
LIN {X 0,Y 343.352,Z 873.001,A -85,B 0,C 180,E1 13303.397,E2 13303.397} C_VEL
LIN {X 0,Y 339.255,Z 885.143,A -85,B 0,C 180,E1 13307.87,E2 13307.87} C_VEL
LIN {X 0,Y 336.658,Z 891.936,A -85,B 0,C 180,E1 13312.267,E2 13312.267} C_VEL
LIN {X 0,Y 335.012,Z 894.391,A -85,B 0,C 180,E1 13317.413,E2 13317.413} C_VEL
LIN {X 0,Y 334.555,Z 891.275,A -85,B 0,C 180,E1 13322.579,E2 13322.579} C_VEL
LIN {X 0,Y 334.925,Z 882.214,A -85,B 0,C 180,E1 13327.762,E2 13327.762} C_VEL
LIN {X 0,Y 336.483,Z 867.472,A -85,B 0,C 180,E1 13332.621,E2 13332.621} C_VEL
LIN {X 0,Y 338.999,Z 847.59,A -85,B 0,C 180,E1 13336.915,E2 13336.915} C_VEL
LIN {X 0,Y 341.993,Z 823.17,A -85,B 0,C 180,E1 13340.494,E2 13340.494} C_VEL
LIN {X 0,Y 344.755,Z 795.881,A -85,B 0,C 180,E1 13343.191,E2 13343.191} C_VEL
LIN {X 0,Y 346.919,Z 764.455,A -85,B 0,C 180,E1 13345.097,E2 13345.097} C_VEL
LIN {X 0,Y 347.505,Z 736.525,A -85,B 0,C 180,E1 13346.129,E2 13346.129} C_VEL
LIN {X 0,Y 329.605,Z 685.03,A -85,B 0,C 180,E1 13349.631,E2 13349.631} C_VEL
LIN {X 0,Y 329.38,Z 685.03,A -85,B 0,C 180,E1 13356.543,E2 13356.543} C_VEL
LIN {X 0,Y 329.406,Z 685.03,A -85,B 0,C 180,E1 13363.392,E2 13363.392} C_VEL
LIN {X 0,Y 329.482,Z 685.219,A -85,B 0,C 180,E1 13369.383,E2 13369.383} C_VEL
LIN {X 0,Y 334.114,Z 694.938,A -85,B 0,C 180,E1 13370.355,E2 13370.355} C_VEL
LIN {X 0,Y 350.033,Z 726.576,A -85,B 0,C 180,E1 13373.526,E2 13373.526} C_VEL
LIN {X 0,Y 359.104,Z 754.332,A -85,B 0,C 180,E1 13376.272,E2 13376.272} C_VEL
LIN {X 0,Y 359.574,Z 761.98,A -85,B 0,C 180,E1 13376.931,E2 13376.931} C_VEL
LIN {X 0,Y 355.221,Z 792.18,A -85,B 0,C 180,E1 13379.522,E2 13379.522} C_VEL
LIN {X 0,Y 349.749,Z 820.184,A -85,B 0,C 180,E1 13383.056,E2 13383.056} C_VEL
LIN {X 0,Y 344.249,Z 843.812,A -85,B 0,C 180,E1 13387.357,E2 13387.357} C_VEL
LIN {X 0,Y 339.322,Z 862.939,A -85,B 0,C 180,E1 13392.436,E2 13392.436} C_VEL
LIN {X 0,Y 336.216,Z 875.941,A -85,B 0,C 180,E1 13397.686,E2 13397.686} C_VEL
LIN {X 0,Y 334.456,Z 883.822,A -85,B 0,C 180,E1 13402.936,E2 13402.936} C_VEL
LIN {X 0,Y 333.846,Z 887.016,A -85,B 0,C 180,E1 13407.405,E2 13407.405} C_VEL
LIN {X 0,Y 333.847,Z 886.981,A -85,B 0,C 180,E1 13412.587,E2 13412.587} C_VEL
LIN {X 0,Y 334.683,Z 882.914,A -85,B 0,C 180,E1 13417.77,E2 13417.77} C_VEL
LIN {X 0,Y 336.837,Z 873.049,A -85,B 0,C 180,E1 13423.6,E2 13423.6} C_VEL
LIN {X 0,Y 340.719,Z 857.661,A -85,B 0,C 180,E1 13429.061,E2 13429.061} C_VEL
LIN {X 0,Y 345.605,Z 838.028,A -85,B 0,C 180,E1 13433.749,E2 13433.749} C_VEL
LIN {X 0,Y 351.205,Z 813.181,A -85,B 0,C 180,E1 13437.854,E2 13437.854} C_VEL
LIN {X 0,Y 356.248,Z 785.458,A -85,B 0,C 180,E1 13441.05,E2 13441.05} C_VEL
LIN {X 0,Y 359.675,Z 757.311,A -85,B 0,C 180,E1 13443.32,E2 13443.32} C_VEL
LIN {X 0,Y 350.647,Z 728.08,A -85,B 0,C 180,E1 13446.222,E2 13446.222} C_VEL
LIN {X 0,Y 334.346,Z 695.362,A -85,B 0,C 180,E1 13449.483,E2 13449.483} C_VEL
LIN {X 0,Y 329.531,Z 686.025,A -85,B 0,C 180,E1 13450.469,E2 13450.469} C_VEL
LIN {X 0,Y 329.428,Z 685.03,A -85,B 0,C 180,E1 13450.61,E2 13450.61} C_VEL
LIN {X 0,Y 329.383,Z 685.03,A -85,B 0,C 180,E1 13457.136,E2 13457.136} C_VEL
LIN {X 0,Y 329.398,Z 685.03,A -85,B 0,C 180,E1 13463.46,E2 13463.46} C_VEL
LIN {X 0,Y 329.63,Z 685.03,A -85,B 0,C 180,E1 13470.432,E2 13470.432} C_VEL
LIN {X 0,Y 329.95,Z 685.03,A -85,B 0,C 180,E1 13478.547,E2 13478.547} C_VEL
LIN {X 0,Y 330.344,Z 685.03,A -85,B 0,C 180,E1 13484.1,E2 13484.1} C_VEL
LIN {X 0,Y 330.765,Z 685.03,A -85,B 0,C 180,E1 13492.14,E2 13492.14} C_VEL
LIN {X 0,Y 331.348,Z 685.03,A -85,B 0,C 180,E1 13500.006,E2 13500.006} C_VEL
LIN {X 0,Y 330.714,Z 685.03,A -85,B 0,C 180,E1 13507.873,E2 13507.873} C_VEL
LIN {X 0,Y 330.227,Z 685.03,A -85,B 0,C 180,E1 13515.917,E2 13515.917} C_VEL
LIN {X 0,Y 329.786,Z 685.03,A -85,B 0,C 180,E1 13524.323,E2 13524.323} C_VEL
LIN {X 0,Y 329.523,Z 685.03,A -85,B 0,C 180,E1 13530.251,E2 13530.251} C_VEL
LIN {X 0,Y 329.601,Z 685.629,A -85,B 0,C 180,E1 13533.861,E2 13533.861} C_VEL
LIN {X 0,Y 336.881,Z 704.516,A -85,B 0,C 180,E1 13536.737,E2 13536.737} C_VEL
LIN {X 0,Y 361.043,Z 755.307,A -85,B 0,C 180,E1 13541.746,E2 13541.746} C_VEL
LIN {X 0,Y 371.9,Z 783.621,A -85,B 0,C 180,E1 13544.424,E2 13544.424} C_VEL
LIN {X 0,Y 365.037,Z 825.746,A -85,B 0,C 180,E1 13546.894,E2 13546.894} C_VEL
LIN {X 0,Y 357.287,Z 863.715,A -85,B 0,C 180,E1 13550.189,E2 13550.189} C_VEL
LIN {X 0,Y 349.399,Z 899.32,A -85,B 0,C 180,E1 13554.511,E2 13554.511} C_VEL
LIN {X 0,Y 342.5,Z 929.668,A -85,B 0,C 180,E1 13559.575,E2 13559.575} C_VEL
LIN {X 0,Y 337.259,Z 954.459,A -85,B 0,C 180,E1 13565.202,E2 13565.202} C_VEL
LIN {X 0,Y 333.757,Z 974.493,A -85,B 0,C 180,E1 13571.553,E2 13571.553} C_VEL
LIN {X 0,Y 332.43,Z 987.484,A -85,B 0,C 180,E1 13577.641,E2 13577.641} C_VEL
LIN {X 0,Y 332.189,Z 994.938,A -85,B 0,C 180,E1 13583.483,E2 13583.483} C_VEL
LIN {X 0,Y 332.135,Z 997.411,A -85,B 0,C 180,E1 13588.276,E2 13588.276} C_VEL
LIN {X 0,Y 332.216,Z 996.89,A -85,B 0,C 180,E1 13592.608,E2 13592.608} C_VEL
LIN {X 0,Y 332.314,Z 992.7,A -85,B 0,C 180,E1 13597.834,E2 13597.834} C_VEL
LIN {X 0,Y 332.761,Z 983.176,A -85,B 0,C 180,E1 13603.778,E2 13603.778} C_VEL
LIN {X 0,Y 334.548,Z 967.066,A -85,B 0,C 180,E1 13610.122,E2 13610.122} C_VEL
LIN {X 0,Y 338.154,Z 945.213,A -85,B 0,C 180,E1 13616.152,E2 13616.152} C_VEL
LIN {X 0,Y 340.989,Z 930.971,A -85,B 0,C 180,E1 13619.252,E2 13619.252} C_VEL
LIN {X 0,Y 339.479,Z 920.166,A -85,B 0,C 180,E1 13621.568,E2 13621.568} C_VEL
LIN {X 0,Y 338.461,Z 908.833,A -85,B 0,C 180,E1 13623.822,E2 13623.822} C_VEL
LIN {X 0,Y 347.566,Z 872.254,A -85,B 0,C 180,E1 13629.136,E2 13629.136} C_VEL
LIN {X 0,Y 358.44,Z 830.712,A -85,B 0,C 180,E1 13633.588,E2 13633.588} C_VEL
LIN {X 0,Y 370.386,Z 786.493,A -85,B 0,C 180,E1 13636.979,E2 13636.979} C_VEL
LIN {X 0,Y 371.541,Z 761.966,A -85,B 0,C 180,E1 13640.258,E2 13640.258} C_VEL
LIN {X 0,Y 371.062,Z 756.824,A -85,B 0,C 180,E1 13641.64,E2 13641.64} C_VEL
LIN {X 0,Y 369.101,Z 755.503,A -85,B 0,C 180,E1 13645.082,E2 13645.082} C_VEL
LIN {X 0,Y 369.029,Z 759.797,A -85,B 0,C 180,E1 13647.536,E2 13647.536} C_VEL
LIN {X 0,Y 368.653,Z 763.116,A -85,B 0,C 180,E1 13648.262,E2 13648.262} C_VEL
LIN {X 0,Y 356.097,Z 805.14,A -85,B 0,C 180,E1 13651.524,E2 13651.524} C_VEL
LIN {X 0,Y 348.537,Z 835.07,A -85,B 0,C 180,E1 13654.857,E2 13654.857} C_VEL
LIN {X 0,Y 342.13,Z 857.411,A -85,B 0,C 180,E1 13658.564,E2 13658.564} C_VEL
LIN {X 0,Y 336.178,Z 875.469,A -85,B 0,C 180,E1 13663.032,E2 13663.032} C_VEL
LIN {X 0,Y 331.829,Z 887.214,A -85,B 0,C 180,E1 13667.595,E2 13667.595} C_VEL
LIN {X 0,Y 329.06,Z 893.695,A -85,B 0,C 180,E1 13672.087,E2 13672.087} C_VEL
LIN {X 0,Y 327.281,Z 895.876,A -85,B 0,C 180,E1 13677.352,E2 13677.352} C_VEL
LIN {X 0,Y 326.756,Z 892.504,A -85,B 0,C 180,E1 13682.641,E2 13682.641} C_VEL
LIN {X 0,Y 327.165,Z 883.219,A -85,B 0,C 180,E1 13687.947,E2 13687.947} C_VEL
LIN {X 0,Y 328.786,Z 868.177,A -85,B 0,C 180,E1 13692.922,E2 13692.922} C_VEL
LIN {X 0,Y 331.305,Z 848.983,A -85,B 0,C 180,E1 13697.132,E2 13697.132} C_VEL
LIN {X 0,Y 334.408,Z 824.588,A -85,B 0,C 180,E1 13700.807,E2 13700.807} C_VEL
LIN {X 0,Y 337.372,Z 796.64,A -85,B 0,C 180,E1 13703.637,E2 13703.637} C_VEL
LIN {X 0,Y 339.595,Z 765.719,A -85,B 0,C 180,E1 13705.553,E2 13705.553} C_VEL
LIN {X 0,Y 340.049,Z 737.614,A -85,B 0,C 180,E1 13706.644,E2 13706.644} C_VEL
LIN {X 0,Y 321.614,Z 685.03,A -85,B 0,C 180,E1 13710.37,E2 13710.37} C_VEL
LIN {X 0,Y 321.451,Z 685.03,A -85,B 0,C 180,E1 13717.597,E2 13717.597} C_VEL
LIN {X 0,Y 321.379,Z 685.03,A -85,B 0,C 180,E1 13725.217,E2 13725.217} C_VEL
LIN {X 0,Y 321.558,Z 685.03,A -85,B 0,C 180,E1 13728.084,E2 13728.084} C_VEL
LIN {X 0,Y 324.069,Z 690.829,A -85,B 0,C 180,E1 13728.693,E2 13728.693} C_VEL
LIN {X 0,Y 342.368,Z 726.017,A -85,B 0,C 180,E1 13732.485,E2 13732.485} C_VEL
LIN {X 0,Y 351.761,Z 753.626,A -85,B 0,C 180,E1 13735.322,E2 13735.322} C_VEL
LIN {X 0,Y 353.084,Z 763.183,A -85,B 0,C 180,E1 13736.242,E2 13736.242} C_VEL
LIN {X 0,Y 348.522,Z 793.406,A -85,B 0,C 180,E1 13738.872,E2 13738.872} C_VEL
LIN {X 0,Y 342.821,Z 821.416,A -85,B 0,C 180,E1 13742.466,E2 13742.466} C_VEL
LIN {X 0,Y 337.003,Z 845.231,A -85,B 0,C 180,E1 13746.886,E2 13746.886} C_VEL
LIN {X 0,Y 331.865,Z 864.218,A -85,B 0,C 180,E1 13752.039,E2 13752.039} C_VEL
LIN {X 0,Y 328.602,Z 877.186,A -85,B 0,C 180,E1 13757.396,E2 13757.396} C_VEL
LIN {X 0,Y 326.474,Z 885.959,A -85,B 0,C 180,E1 13763.666,E2 13763.666} C_VEL
LIN {X 0,Y 325.995,Z 888.782,A -85,B 0,C 180,E1 13769.996,E2 13769.996} C_VEL
LIN {X 0,Y 326.557,Z 885.752,A -85,B 0,C 180,E1 13776.466,E2 13776.466} C_VEL
LIN {X 0,Y 328.608,Z 877.014,A -85,B 0,C 180,E1 13782.595,E2 13782.595} C_VEL
LIN {X 0,Y 332.017,Z 863.701,A -85,B 0,C 180,E1 13788.018,E2 13788.018} C_VEL
LIN {X 0,Y 337.152,Z 844.517,A -85,B 0,C 180,E1 13793.167,E2 13793.167} C_VEL
LIN {X 0,Y 342.906,Z 820.862,A -85,B 0,C 180,E1 13797.518,E2 13797.518} C_VEL
LIN {X 0,Y 348.343,Z 794.069,A -85,B 0,C 180,E1 13800.956,E2 13800.956} C_VEL
LIN {X 0,Y 353.06,Z 763.001,A -85,B 0,C 180,E1 13803.666,E2 13803.666} C_VEL
LIN {X 0,Y 348.482,Z 742.56,A -85,B 0,C 180,E1 13805.733,E2 13805.733} C_VEL
LIN {X 0,Y 336.876,Z 714.269,A -85,B 0,C 180,E1 13808.598,E2 13808.598} C_VEL
LIN {X 0,Y 321.472,Z 685.777,A -85,B 0,C 180,E1 13811.76,E2 13811.76} C_VEL
LIN {X 0,Y 321.364,Z 685.03,A -85,B 0,C 180,E1 13818.912,E2 13818.912} C_VEL
LIN {X 0,Y 321.477,Z 685.03,A -85,B 0,C 180,E1 13825.728,E2 13825.728} C_VEL
LIN {X 0,Y 321.768,Z 685.03,A -85,B 0,C 180,E1 13833.002,E2 13833.002} C_VEL
LIN {X 0,Y 322.16,Z 685.03,A -85,B 0,C 180,E1 13840.868,E2 13840.868} C_VEL
LIN {X 0,Y 322.588,Z 685.03,A -85,B 0,C 180,E1 13846.481,E2 13846.481} C_VEL
LIN {X 0,Y 323.026,Z 685.03,A -85,B 0,C 180,E1 13854.646,E2 13854.646} C_VEL
LIN {X 0,Y 323.444,Z 685.03,A -85,B 0,C 180,E1 13860.006,E2 13860.006} C_VEL
LIN {X 0,Y 322.774,Z 685.03,A -85,B 0,C 180,E1 13868.068,E2 13868.068} C_VEL
LIN {X 0,Y 322.276,Z 685.03,A -85,B 0,C 180,E1 13876.321,E2 13876.321} C_VEL
LIN {X 0,Y 321.981,Z 685.03,A -85,B 0,C 180,E1 13882.024,E2 13882.024} C_VEL
LIN {X 0,Y 321.682,Z 685.03,A -85,B 0,C 180,E1 13887.98,E2 13887.98} C_VEL
LIN {X 0,Y 321.62,Z 685.691,A -85,B 0,C 180,E1 13892.75,E2 13892.75} C_VEL
LIN {X 0,Y 328.743,Z 703.799,A -85,B 0,C 180,E1 13895.576,E2 13895.576} C_VEL
LIN {X 0,Y 353.253,Z 755.239,A -85,B 0,C 180,E1 13900.855,E2 13900.855} C_VEL
LIN {X 0,Y 364.929,Z 787.209,A -85,B 0,C 180,E1 13903.938,E2 13903.938} C_VEL
LIN {X 0,Y 357.791,Z 827.424,A -85,B 0,C 180,E1 13906.415,E2 13906.415} C_VEL
LIN {X 0,Y 349.697,Z 865.433,A -85,B 0,C 180,E1 13909.836,E2 13909.836} C_VEL
LIN {X 0,Y 342.013,Z 899.01,A -85,B 0,C 180,E1 13914.033,E2 13914.033} C_VEL
LIN {X 0,Y 335.036,Z 928.783,A -85,B 0,C 180,E1 13919.103,E2 13919.103} C_VEL
LIN {X 0,Y 329.505,Z 953.918,A -85,B 0,C 180,E1 13924.94,E2 13924.94} C_VEL
LIN {X 0,Y 326.028,Z 972.971,A -85,B 0,C 180,E1 13931.099,E2 13931.099} C_VEL
LIN {X 0,Y 324.589,Z 986.421,A -85,B 0,C 180,E1 13937.501,E2 13937.501} C_VEL
LIN {X 0,Y 324.352,Z 993.71,A -85,B 0,C 180,E1 13943.325,E2 13943.325} C_VEL
LIN {X 0,Y 324.337,Z 996.026,A -85,B 0,C 180,E1 13947.337,E2 13947.337} C_VEL
LIN {X 0,Y 324.387,Z 995.709,A -85,B 0,C 180,E1 13952.67,E2 13952.67} C_VEL
LIN {X 0,Y 324.485,Z 991.485,A -85,B 0,C 180,E1 13958.024,E2 13958.024} C_VEL
LIN {X 0,Y 324.923,Z 981.887,A -85,B 0,C 180,E1 13964.117,E2 13964.117} C_VEL
LIN {X 0,Y 326.852,Z 965.684,A -85,B 0,C 180,E1 13970.617,E2 13970.617} C_VEL
LIN {X 0,Y 330.725,Z 943.792,A -85,B 0,C 180,E1 13976.786,E2 13976.786} C_VEL
LIN {X 0,Y 337.112,Z 914.519,A -85,B 0,C 180,E1 13982.839,E2 13982.839} C_VEL
LIN {X 0,Y 338.461,Z 908.833,A -85,B 0,C 180,E1 13983.822,E2 13983.822} C_VEL
LIN {X 0,Y 337.721,Z 897.214,A -85,B 0,C 180,E1 13986.05,E2 13986.05} C_VEL
LIN {X 0,Y 337.508,Z 885.124,A -85,B 0,C 180,E1 13988.196,E2 13988.196} C_VEL
LIN {X 0,Y 349.224,Z 843.8,A -85,B 0,C 180,E1 13993.259,E2 13993.259} C_VEL
LIN {X 0,Y 362.576,Z 798.796,A -85,B 0,C 180,E1 13997.192,E2 13997.192} C_VEL
LIN {X 0,Y 365.388,Z 788.183,A -85,B 0,C 180,E1 13998.028,E2 13998.028} C_VEL
LIN {X 0,Y 367.782,Z 765.893,A -85,B 0,C 180,E1 14001.23,E2 14001.23} C_VEL
LIN {X 0,Y 367.55,Z 763.658,A -85,B 0,C 180,E1 14001.985,E2 14001.985} C_VEL
LIN {X 0,Y 365.908,Z 762.632,A -85,B 0,C 180,E1 14004.732,E2 14004.732} C_VEL
LIN {X 0,Y 365.431,Z 766.629,A -85,B 0,C 180,E1 14007.218,E2 14007.218} C_VEL
LIN {X 0,Y 350.983,Z 808.971,A -85,B 0,C 180,E1 14010.718,E2 14010.718} C_VEL
LIN {X 0,Y 342.455,Z 838.424,A -85,B 0,C 180,E1 14014.202,E2 14014.202} C_VEL
LIN {X 0,Y 335.321,Z 860.643,A -85,B 0,C 180,E1 14018.107,E2 14018.107} C_VEL
LIN {X 0,Y 329.035,Z 878.012,A -85,B 0,C 180,E1 14022.652,E2 14022.652} C_VEL
LIN {X 0,Y 324.292,Z 889.534,A -85,B 0,C 180,E1 14027.444,E2 14027.444} C_VEL
LIN {X 0,Y 321.456,Z 895.467,A -85,B 0,C 180,E1 14031.899,E2 14031.899} C_VEL
LIN {X 0,Y 319.531,Z 897.365,A -85,B 0,C 180,E1 14037.287,E2 14037.287} C_VEL
LIN {X 0,Y 318.963,Z 893.711,A -85,B 0,C 180,E1 14042.705,E2 14042.705} C_VEL
LIN {X 0,Y 319.388,Z 884.173,A -85,B 0,C 180,E1 14048.142,E2 14048.142} C_VEL
LIN {X 0,Y 321.115,Z 868.864,A -85,B 0,C 180,E1 14053.236,E2 14053.236} C_VEL
LIN {X 0,Y 323.808,Z 848.915,A -85,B 0,C 180,E1 14057.636,E2 14057.636} C_VEL
LIN {X 0,Y 327.131,Z 823.25,A -85,B 0,C 180,E1 14061.47,E2 14061.47} C_VEL
LIN {X 0,Y 330.162,Z 794.951,A -85,B 0,C 180,E1 14064.281,E2 14064.281} C_VEL
LIN {X 0,Y 332.466,Z 763.036,A -85,B 0,C 180,E1 14066.204,E2 14066.204} C_VEL
LIN {X 0,Y 332.951,Z 739.827,A -85,B 0,C 180,E1 14067.109,E2 14067.109} C_VEL
LIN {X 0,Y 314.696,Z 688.945,A -85,B 0,C 180,E1 14070.847,E2 14070.847} C_VEL
LIN {X 0,Y 313.621,Z 685.03,A -85,B 0,C 180,E1 14071.19,E2 14071.19} C_VEL
LIN {X 0,Y 313.402,Z 685.03,A -85,B 0,C 180,E1 14078.739,E2 14078.739} C_VEL
LIN {X 0,Y 313.628,Z 685.708,A -85,B 0,C 180,E1 14086.773,E2 14086.773} C_VEL
LIN {X 0,Y 335.333,Z 727.012,A -85,B 0,C 180,E1 14091.541,E2 14091.541} C_VEL
LIN {X 0,Y 344.889,Z 754.717,A -85,B 0,C 180,E1 14094.513,E2 14094.513} C_VEL
LIN {X 0,Y 346.482,Z 765.892,A -85,B 0,C 180,E1 14095.634,E2 14095.634} C_VEL
LIN {X 0,Y 341.591,Z 796.093,A -85,B 0,C 180,E1 14098.353,E2 14098.353} C_VEL
LIN {X 0,Y 335.793,Z 823.153,A -85,B 0,C 180,E1 14101.931,E2 14101.931} C_VEL
LIN {X 0,Y 329.714,Z 846.921,A -85,B 0,C 180,E1 14106.461,E2 14106.461} C_VEL
LIN {X 0,Y 324.612,Z 864.947,A -85,B 0,C 180,E1 14111.447,E2 14111.447} C_VEL
LIN {X 0,Y 320.963,Z 878.436,A -85,B 0,C 180,E1 14117.091,E2 14117.091} C_VEL
LIN {X 0,Y 319.209,Z 885.514,A -85,B 0,C 180,E1 14121.842,E2 14121.842} C_VEL
LIN {X 0,Y 318.275,Z 889.509,A -85,B 0,C 180,E1 14127.278,E2 14127.278} C_VEL
LIN {X 0,Y 318.277,Z 889.474,A -85,B 0,C 180,E1 14132.714,E2 14132.714} C_VEL
LIN {X 0,Y 319.22,Z 885.412,A -85,B 0,C 180,E1 14138.149,E2 14138.149} C_VEL
LIN {X 0,Y 321.667,Z 875.548,A -85,B 0,C 180,E1 14144.254,E2 14144.254} C_VEL
LIN {X 0,Y 325.994,Z 860.156,A -85,B 0,C 180,E1 14149.958,E2 14149.958} C_VEL
LIN {X 0,Y 331.478,Z 840.195,A -85,B 0,C 180,E1 14154.901,E2 14154.901} C_VEL
LIN {X 0,Y 337.445,Z 815.898,A -85,B 0,C 180,E1 14159.056,E2 14159.056} C_VEL
LIN {X 0,Y 343.152,Z 787.07,A -85,B 0,C 180,E1 14162.474,E2 14162.474} C_VEL
LIN {X 0,Y 346.313,Z 761.264,A -85,B 0,C 180,E1 14164.666,E2 14164.666} C_VEL
LIN {X 0,Y 337.866,Z 733.159,A -85,B 0,C 180,E1 14167.702,E2 14167.702} C_VEL
LIN {X 0,Y 322.477,Z 701.884,A -85,B 0,C 180,E1 14171.118,E2 14171.118} C_VEL
LIN {X 0,Y 313.574,Z 685.672,A -85,B 0,C 180,E1 14173.114,E2 14173.114} C_VEL
LIN {X 0,Y 313.386,Z 685.03,A -85,B 0,C 180,E1 14181.258,E2 14181.258} C_VEL
LIN {X 0,Y 313.6,Z 685.03,A -85,B 0,C 180,E1 14188.052,E2 14188.052} C_VEL
LIN {X 0,Y 313.891,Z 685.03,A -85,B 0,C 180,E1 14195.977,E2 14195.977} C_VEL
LIN {X 0,Y 314.51,Z 685.03,A -85,B 0,C 180,E1 14203.651,E2 14203.651} C_VEL
